// TwinCAT 3 PLC project _7000_Theresianum
// ProgramVersion: 3.1.4024.0
// libraries:
//   EfficientIO Communicator, * (EfficientIO)
//   EfficientIO ModbusTCP, * (EfficientIO)
//   Lynus Energy Basic, * (Lynus AG)
//   Lynus Persistent Data V1, * (Lynus AG)
//   Lynus Standards, * (Lynus AG)
//   Tc2_BABasic, * (Beckhoff Automation GmbH)
//   Tc2_Standard, * (Beckhoff Automation GmbH)
//   Tc2_System, * (Beckhoff Automation GmbH)
//   Tc2_Utilities, * (Beckhoff Automation GmbH)
//   Tc3_IotBase, * (Beckhoff Automation GmbH)
//   Tc3_JsonXml, * (Beckhoff Automation GmbH)
//   Tc3_Module, * (Beckhoff Automation GmbH)
// project tree:
//   / FastTask.TcTTO, MiddleTask.TcTTO, SlowTask.TcTTO
//   FBs/ FB_EM_Beckhoff_KL3403.TcPOU, FB_MqttCommunicator_V2_1.TcPOU, FB_Shelly_Pro.TcPOU (not stored), FB_Shelly_Pro1PM_Helper.TcPOU, FB_Shelly_Pro3EM.TcPOU, FB_Shelly_Pro3EM_Helper.TcPOU
//   POUs/ prgComEffIO.TcPOU, prgEM.TcPOU, prgPersistent.TcPOU, prgRWEffIO.TcPOU (not stored), prgShelly.TcPOU, prgVarEffIO.TcPOU (not stored), prg_SystemTime.TcPOU (not stored)
// real-time tasks:
//   TASK FastTask: cycle T#5ms, priority 6, ADS port 350
//   TASK MiddleTask: cycle T#10ms, priority 8, ADS port 351
//   TASK SlowTask: cycle T#20ms, priority 10, ADS port 352
// I/O:
//   DEVICE Gerät 1 (Beckhoff CCAT)
//   DEVICE Gerät 2 (CX-BK)
//     Box 1 (CX-BK)
// variable links:
//   (this object) <-> Device 2 (CX-BK)/Box 1 (CX-BK)
//     MiddleTask Inputs/prgEM.fbEM1.fbKL3403.byStateCH1 <-> Term 2 (KL3403)/Channel 1/Status
//     MiddleTask Inputs/prgEM.fbEM1.fbKL3403.byStateCH2 <-> Term 2 (KL3403)/Channel 2/Status
//     MiddleTask Inputs/prgEM.fbEM1.fbKL3403.byStateCH3 <-> Term 2 (KL3403)/Channel 3/Status
//     MiddleTask Inputs/prgEM.fbEM2.fbKL3403.byStateCH1 <-> Term 3 (KL3403)/Channel 1/Status
//     MiddleTask Inputs/prgEM.fbEM2.fbKL3403.byStateCH2 <-> Term 3 (KL3403)/Channel 2/Status
//     MiddleTask Inputs/prgEM.fbEM2.fbKL3403.byStateCH3 <-> Term 3 (KL3403)/Channel 3/Status
//     MiddleTask Inputs/prgEM.fbEM3.fbKL3403.byStateCH1 <-> Term 4 (KL3403)/Channel 1/Status
//     MiddleTask Inputs/prgEM.fbEM3.fbKL3403.byStateCH2 <-> Term 4 (KL3403)/Channel 2/Status
//     MiddleTask Inputs/prgEM.fbEM3.fbKL3403.byStateCH3 <-> Term 4 (KL3403)/Channel 3/Status
//     MiddleTask Inputs/prgEM.fbEM4.fbKL3403.byStateCH1 <-> Term 5 (KL3403)/Channel 1/Status
//     MiddleTask Inputs/prgEM.fbEM4.fbKL3403.byStateCH2 <-> Term 5 (KL3403)/Channel 2/Status
//     MiddleTask Inputs/prgEM.fbEM4.fbKL3403.byStateCH3 <-> Term 5 (KL3403)/Channel 3/Status
//     MiddleTask Inputs/prgEM.fbEM5.fbKL3403.byStateCH1 <-> Term 6 (KL3403)/Channel 1/Status
//     MiddleTask Inputs/prgEM.fbEM5.fbKL3403.byStateCH2 <-> Term 6 (KL3403)/Channel 2/Status
//     MiddleTask Inputs/prgEM.fbEM5.fbKL3403.byStateCH3 <-> Term 6 (KL3403)/Channel 3/Status
//     MiddleTask Inputs/prgEM.fbEM1.fbKL3403.iDataInCH1 <-> Term 2 (KL3403)/Channel 1/Daten Ein
//     MiddleTask Inputs/prgEM.fbEM1.fbKL3403.iDataInCH2 <-> Term 2 (KL3403)/Channel 2/Daten Ein
//     MiddleTask Inputs/prgEM.fbEM1.fbKL3403.iDataInCH3 <-> Term 2 (KL3403)/Channel 3/Daten Ein
//     MiddleTask Inputs/prgEM.fbEM2.fbKL3403.iDataInCH1 <-> Term 3 (KL3403)/Channel 1/Daten Ein
//     MiddleTask Inputs/prgEM.fbEM2.fbKL3403.iDataInCH2 <-> Term 3 (KL3403)/Channel 2/Daten Ein
//     MiddleTask Inputs/prgEM.fbEM2.fbKL3403.iDataInCH3 <-> Term 3 (KL3403)/Channel 3/Daten Ein
//     MiddleTask Inputs/prgEM.fbEM3.fbKL3403.iDataInCH1 <-> Term 4 (KL3403)/Channel 1/Daten Ein
//     MiddleTask Inputs/prgEM.fbEM3.fbKL3403.iDataInCH2 <-> Term 4 (KL3403)/Channel 2/Daten Ein
//     MiddleTask Inputs/prgEM.fbEM3.fbKL3403.iDataInCH3 <-> Term 4 (KL3403)/Channel 3/Daten Ein
//     MiddleTask Inputs/prgEM.fbEM4.fbKL3403.iDataInCH1 <-> Term 5 (KL3403)/Channel 1/Daten Ein
//     MiddleTask Inputs/prgEM.fbEM4.fbKL3403.iDataInCH2 <-> Term 5 (KL3403)/Channel 2/Daten Ein
//     MiddleTask Inputs/prgEM.fbEM4.fbKL3403.iDataInCH3 <-> Term 5 (KL3403)/Channel 3/Daten Ein
//     MiddleTask Inputs/prgEM.fbEM5.fbKL3403.iDataInCH1 <-> Term 6 (KL3403)/Channel 1/Daten Ein
//     MiddleTask Inputs/prgEM.fbEM5.fbKL3403.iDataInCH2 <-> Term 6 (KL3403)/Channel 2/Daten Ein
//     MiddleTask Inputs/prgEM.fbEM5.fbKL3403.iDataInCH3 <-> Term 6 (KL3403)/Channel 3/Daten Ein
//     MiddleTask Outputs/prgEM.fbEM1.fbKL3403.byCntrCH1 <-> Term 2 (KL3403)/Channel 1/Kontrolle
//     MiddleTask Outputs/prgEM.fbEM1.fbKL3403.byCntrCH2 <-> Term 2 (KL3403)/Channel 2/Kontrolle
//     MiddleTask Outputs/prgEM.fbEM1.fbKL3403.byCntrCH3 <-> Term 2 (KL3403)/Channel 3/Kontrolle
//     MiddleTask Outputs/prgEM.fbEM2.fbKL3403.byCntrCH1 <-> Term 3 (KL3403)/Channel 1/Kontrolle
//     MiddleTask Outputs/prgEM.fbEM2.fbKL3403.byCntrCH2 <-> Term 3 (KL3403)/Channel 2/Kontrolle
//     MiddleTask Outputs/prgEM.fbEM2.fbKL3403.byCntrCH3 <-> Term 3 (KL3403)/Channel 3/Kontrolle
//     MiddleTask Outputs/prgEM.fbEM3.fbKL3403.byCntrCH1 <-> Term 4 (KL3403)/Channel 1/Kontrolle
//     MiddleTask Outputs/prgEM.fbEM3.fbKL3403.byCntrCH2 <-> Term 4 (KL3403)/Channel 2/Kontrolle
//     MiddleTask Outputs/prgEM.fbEM3.fbKL3403.byCntrCH3 <-> Term 4 (KL3403)/Channel 3/Kontrolle
//     MiddleTask Outputs/prgEM.fbEM4.fbKL3403.byCntrCH1 <-> Term 5 (KL3403)/Channel 1/Kontrolle
//     MiddleTask Outputs/prgEM.fbEM4.fbKL3403.byCntrCH2 <-> Term 5 (KL3403)/Channel 2/Kontrolle
//     MiddleTask Outputs/prgEM.fbEM4.fbKL3403.byCntrCH3 <-> Term 5 (KL3403)/Channel 3/Kontrolle
//     MiddleTask Outputs/prgEM.fbEM5.fbKL3403.byCntrCH1 <-> Term 6 (KL3403)/Channel 1/Kontrolle
//     MiddleTask Outputs/prgEM.fbEM5.fbKL3403.byCntrCH2 <-> Term 6 (KL3403)/Channel 2/Kontrolle
//     MiddleTask Outputs/prgEM.fbEM5.fbKL3403.byCntrCH3 <-> Term 6 (KL3403)/Channel 3/Kontrolle

CONFIGURATION _7000_Theresianum
    RESOURCE PLC ON TwinCAT3
        TASK FastTask(INTERVAL := T#5ms, PRIORITY := 6);
        TASK MiddleTask(INTERVAL := T#10ms, PRIORITY := 8);
        TASK SlowTask(INTERVAL := T#20ms, PRIORITY := 10);
        PROGRAM prgVarEffIO WITH FastTask : prgVarEffIO;
        PROGRAM prgRWEffIO WITH FastTask : prgRWEffIO;
        PROGRAM prgPersistent WITH MiddleTask : prgPersistent;
        PROGRAM prgEM WITH MiddleTask : prgEM;
        PROGRAM prgShelly WITH MiddleTask : prgShelly;
        PROGRAM prgComEffIO WITH SlowTask : prgComEffIO;
    END_RESOURCE
END_CONFIGURATION

// ---- POUs/prgPersistent.TcPOU
PROGRAM prgPersistent
VAR
	fbUSV		: FB_WritePersistentData_CX81xx;
	fb_Reboot		: NT_reboot;
	m_Reboot		: BOOL:=FALSE;
END_VAR

fbUSV(
	eSaveModeData:= eUSVSaveMode.eSaveWhenPowerfail, 
	bLoadPersistentDataOk=> , 
	bPowerFailDetect=> , 
	bError=> , 
	bySaveProcess=> , 
	dwStorageLast24h=> , 
	udiErrorCode=> );
(*	
prg_SystemTime();

		
fb_Reboot(	netid := '',
			delay := 2,
			start := m_Reboot);
			
*)

END_PROGRAM

// ---- POUs/prgEM.TcPOU
PROGRAM prgEM
VAR
	fbKBusState					: FB_K_Bus_State;
	fbEM1						: FB_EM_Beckhoff_KL3403;			//Messung 1 Rest
	fbEM1Counter				: FB_EnergyCounter;
	fbEM2						: FB_EM_Beckhoff_KL3403;			//Messung 2 Schulküche
	fbEM2Counter				: FB_EnergyCounter;
	fbEM3						: FB_EM_Beckhoff_KL3403;			//Messung 3 Aufzüge
	fbEM3Counter				: FB_EnergyCounter;
	fbEM4						: FB_EM_Beckhoff_KL3403;			//Messung 4 Heizungsverteiler
	fbEM4Counter				: FB_EnergyCounter;
	fbEM5						: FB_EM_Beckhoff_KL3403;			//Messung 5 Verteiler 14 gesamt
	fbEM5Counter				: FB_EnergyCounter;
	
	lrPowerEM1_1				: LREAL;							//{#lynus.ag#()}
	lrPowerEM1_2				: LREAL;							//{#lynus.ag#()}
	lrPowerEM1_3				: LREAL;							//{#lynus.ag#()}
	lrPowerEM2_1				: LREAL;							//{#lynus.ag#()}
	lrPowerEM2_2				: LREAL;							//{#lynus.ag#()}
	lrPowerEM2_3				: LREAL;							//{#lynus.ag#()}
	lrPowerEM3_1				: LREAL;							//{#lynus.ag#()}
	lrPowerEM3_2				: LREAL;							//{#lynus.ag#()}
	lrPowerEM3_3				: LREAL;							//{#lynus.ag#()}
	lrPowerEM4_1				: LREAL;							//{#lynus.ag#()}
	lrPowerEM4_2				: LREAL;							//{#lynus.ag#()}
	lrPowerEM4_3				: LREAL;							//{#lynus.ag#()}
	lrPowerEM5_1				: LREAL;							//{#lynus.ag#()}
	lrPowerEM5_2				: LREAL;							//{#lynus.ag#()}
	lrPowerEM5_3				: LREAL;							//{#lynus.ag#()}
	
	lrPowerEM1_Total			: LREAL;							//{#lynus.ag#()}
	lrPowerEM2_Total			: LREAL;							//{#lynus.ag#()}
	lrPowerEM3_Total			: LREAL;							//{#lynus.ag#()}
	lrPowerEM4_Total			: LREAL;							//{#lynus.ag#()}
	lrPowerEM5_Total			: LREAL;							//{#lynus.ag#()}
	
	lrCounterGridCon			: LREAL;							
	//lrCounterGridProd			: LREAL;							
	
	lr_GridVoltage1_L1N_V		: LREAL;						
	lr_GridVoltage1_L2N_V		: LREAL;						
	lr_GridVoltage1_L3N_V		: LREAL;						
	lr_GridVoltage2_L1N_V		: LREAL;						
	lr_GridVoltage2_L2N_V		: LREAL;						
	lr_GridVoltage2_L3N_V		: LREAL;						
	lr_GridVoltage3_L1N_V		: LREAL;						
	lr_GridVoltage3_L2N_V		: LREAL;						
	lr_GridVoltage3_L3N_V		: LREAL;						
	lr_GridVoltage4_L1N_V		: LREAL;						
	lr_GridVoltage4_L2N_V		: LREAL;						
	lr_GridVoltage4_L3N_V		: LREAL;						
	lr_GridVoltage5_L1N_V		: LREAL;						
	lr_GridVoltage5_L2N_V		: LREAL;						
	lr_GridVoltage5_L3N_V		: LREAL;						

	lrReactivePowerGrid			: LREAL;							
	lrApparentPowerGrid			: LREAL;							
	
	lrPowerGrid					: LREAL;							//{#lynus.ag#()}

	lrPowerHouse				: LREAL;							//{#lynus.ag#()}
	tmp	: LREAL;
	tmp2	: LREAL;
END_VAR

VAR PERSISTENT
	
	lrCounterEM1					: LREAL;							//{#lynus.ag#()}
	lrCounterEM2					: LREAL;							//{#lynus.ag#()}
	lrCounterEM3					: LREAL;							//{#lynus.ag#()}
	lrCounterEM4					: LREAL;							//{#lynus.ag#()}
	lrCounterEM5					: LREAL;							//{#lynus.ag#()}

END_VAR

//The mapping of this function must be linked with the K-Bus State in the E/A Part
fbKBusState(	uiKBusState_OUT=> , 
				b_Kbus_notOk=> , 
				word_ErrorCount=> );
				
//The mapping of this function must be linked with the KL3403 in the E/A Part

fbEM1(										//Rest
	bEnable:= TRUE, 
	bChannel1Invers:= FALSE,				//Invert power data when transformer are mounted upside down
	bChannel2Invers:= FALSE,
	bChannel3Invers:= FALSE,
	uiCurrentTransformerRatioL1:= 400, 		//Transformer ratio on the secondary side
	uiCurrentTransformerRatioL2:= 400, 
	uiCurrentTransformerRatioL3:= 400, 
	uiKBusState_IN:= fbKBusState.uiKBusState_OUT, 
	stDataEMPower=> , 
	stDataEMCounter=> , 
	stDataEMPowerRealTime=> , 
	stDataEMCounterRealTime=> , 
	diNrOfEM_OUT=> );
	


fbEM2(										// Heizungsverteiler
	bEnable:= TRUE, 
	bChannel1Invers:= FALSE,				//Invert power data when transformer are mounted upside down
	bChannel2Invers:= FALSE,
	bChannel3Invers:= FALSE,	
	uiCurrentTransformerRatioL1:= 400, 		//Transformer ratio on the secondary side
	uiCurrentTransformerRatioL2:= 400, 
	uiCurrentTransformerRatioL3:= 400, 
	uiKBusState_IN:= fbKBusState.uiKBusState_OUT, 
	stDataEMPower=> , 
	stDataEMCounter=> , 
	stDataEMPowerRealTime=> , 
	stDataEMCounterRealTime=> , 
	diNrOfEM_OUT=> );
	
fbEM3(										// Aufzüge
	bEnable:= TRUE, 
	bChannel1Invers:= FALSE,				//Invert power data when transformer are mounted upside down
	bChannel2Invers:= FALSE,
	bChannel3Invers:= FALSE,
	uiCurrentTransformerRatioL1:= 300, 		//Transformer ratio on the secondary side
	uiCurrentTransformerRatioL2:= 300, 
	uiCurrentTransformerRatioL3:= 300, 
	uiKBusState_IN:= fbKBusState.uiKBusState_OUT, 
	stDataEMPower=> , 
	stDataEMCounter=> , 
	stDataEMPowerRealTime=> , 
	stDataEMCounterRealTime=> , 
	diNrOfEM_OUT=> );
	
fbEM4(										// Turnsaal
	bEnable:= TRUE, 
	bChannel1Invers:= FALSE,				//Invert power data when transformer are mounted upside down
	bChannel2Invers:= FALSE,
	bChannel3Invers:= FALSE,
	uiCurrentTransformerRatioL1:= 300, 		//Transformer ratio on the secondary side
	uiCurrentTransformerRatioL2:= 300, 
	uiCurrentTransformerRatioL3:= 300, 
	uiKBusState_IN:= fbKBusState.uiKBusState_OUT, 
	stDataEMPower=> , 
	stDataEMCounter=> , 
	stDataEMPowerRealTime=> , 
	stDataEMCounterRealTime=> , 
	diNrOfEM_OUT=> );
	
fbEM5(										// Verteiler Schulküchen (4x185mm2)
	bEnable:= TRUE, 
	bChannel1Invers:= FALSE,				//Invert power data when transformer are mounted upside down
	bChannel2Invers:= FALSE,
	bChannel3Invers:= FALSE,
	uiCurrentTransformerRatioL1:= 400, 		//Transformer ratio on the secondary side
	uiCurrentTransformerRatioL2:= 400, 
	uiCurrentTransformerRatioL3:= 400, 
	uiKBusState_IN:= fbKBusState.uiKBusState_OUT, 
	stDataEMPower=> , 
	stDataEMCounter=> , 
	stDataEMPowerRealTime=> , 
	stDataEMCounterRealTime=> , 
	diNrOfEM_OUT=> );

//lrCounterGridProd := fbEM1.stDataEMCounter.lrTotalCounterEnergy_Production;	

lrPowerEM1_1 := fbEM1.stDataEMPower.lrPowerL1;
lrPowerEM1_2 := fbEM1.stDataEMPower.lrPowerL2;
lrPowerEM1_3 := fbEM1.stDataEMPower.lrPowerL3;

lrPowerEM1_Total := fbEM1.stDataEMPower.lrPowerTotal;

lrReactivePowerGrid:=fbEM1.stDataEMPower.lrReactivePowerTotal;
lrApparentPowerGrid:=fbEM1.stDataEMPower.lrApparentPowerTotal;

lr_GridVoltage1_L1N_V:=fbEM1.stDataEMPower.lrVoltageL1N;
lr_GridVoltage1_L2N_V:=fbEM1.stDataEMPower.lrVoltageL2N;
lr_GridVoltage1_L3N_V:=fbEM1.stDataEMPower.lrVoltageL3N;

lrPowerEM2_1 := fbEM2.stDataEMPower.lrPowerL1;
lrPowerEM2_2 := fbEM2.stDataEMPower.lrPowerL2;
lrPowerEM2_3 := fbEM2.stDataEMPower.lrPowerL3;

lrPowerEM2_Total := fbEM2.stDataEMPower.lrPowerTotal;

lrReactivePowerGrid:=fbEM2.stDataEMPower.lrReactivePowerTotal;
lrApparentPowerGrid:=fbEM2.stDataEMPower.lrApparentPowerTotal;

lr_GridVoltage2_L1N_V:=fbEM2.stDataEMPower.lrVoltageL1N;
lr_GridVoltage2_L2N_V:=fbEM2.stDataEMPower.lrVoltageL2N;
lr_GridVoltage2_L3N_V:=fbEM2.stDataEMPower.lrVoltageL3N;

lrPowerEM3_1 := fbEM3.stDataEMPower.lrPowerL1;
lrPowerEM3_2 := fbEM3.stDataEMPower.lrPowerL2;
lrPowerEM3_3 := fbEM3.stDataEMPower.lrPowerL3;

lrPowerEM3_Total := fbEM3.stDataEMPower.lrPowerTotal;

lrReactivePowerGrid:=fbEM3.stDataEMPower.lrReactivePowerTotal;
lrApparentPowerGrid:=fbEM3.stDataEMPower.lrApparentPowerTotal;

lr_GridVoltage3_L1N_V:=fbEM3.stDataEMPower.lrVoltageL1N;
lr_GridVoltage3_L2N_V:=fbEM3.stDataEMPower.lrVoltageL2N;
lr_GridVoltage3_L3N_V:=fbEM3.stDataEMPower.lrVoltageL3N;

lrPowerEM4_1 := fbEM4.stDataEMPower.lrPowerL1;
lrPowerEM4_2 := fbEM4.stDataEMPower.lrPowerL2;
lrPowerEM4_3 := fbEM4.stDataEMPower.lrPowerL3;

lrPowerEM4_Total := fbEM4.stDataEMPower.lrPowerTotal;

lrReactivePowerGrid:=fbEM4.stDataEMPower.lrReactivePowerTotal;
lrApparentPowerGrid:=fbEM4.stDataEMPower.lrApparentPowerTotal;

lr_GridVoltage4_L1N_V:=fbEM4.stDataEMPower.lrVoltageL1N;
lr_GridVoltage4_L2N_V:=fbEM4.stDataEMPower.lrVoltageL2N;
lr_GridVoltage4_L3N_V:=fbEM4.stDataEMPower.lrVoltageL3N;

lrPowerEM5_1 := fbEM5.stDataEMPower.lrPowerL1;
lrPowerEM5_2 := fbEM5.stDataEMPower.lrPowerL2;
lrPowerEM5_3 := fbEM5.stDataEMPower.lrPowerL3;

lrPowerEM5_Total := fbEM5.stDataEMPower.lrPowerTotal;

lrReactivePowerGrid:=fbEM5.stDataEMPower.lrReactivePowerTotal;
lrApparentPowerGrid:=fbEM5.stDataEMPower.lrApparentPowerTotal;

lr_GridVoltage5_L1N_V:=fbEM5.stDataEMPower.lrVoltageL1N;
lr_GridVoltage5_L2N_V:=fbEM5.stDataEMPower.lrVoltageL2N;
lr_GridVoltage5_L3N_V:=fbEM5.stDataEMPower.lrVoltageL3N;

lrPowerGrid := LIMIT((fbEM1.stDataEMPower.lrPowerTotal + fbEM2.stDataEMPower.lrPowerTotal + fbEM3.stDataEMPower.lrPowerTotal + fbEM4.stDataEMPower.lrPowerTotal + fbEM5.stDataEMPower.lrPowerTotal),(fbEM1.stDataEMPower.lrPowerTotal + fbEM5.stDataEMPower.lrPowerTotal),999999);
tmp := fbEM1.stDataEMPower.lrPowerTotal + fbEM2.stDataEMPower.lrPowerTotal + fbEM3.stDataEMPower.lrPowerTotal + fbEM4.stDataEMPower.lrPowerTotal + fbEM5.stDataEMPower.lrPowerTotal;
tmp2 := fbEM1.stDataEMPower.lrPowerTotal + fbEM5.stDataEMPower.lrPowerTotal;

lrPowerHouse :=  lrPowerEM1_Total - (lrPowerEM2_Total + lrPowerEM3_Total + lrPowerEM4_Total);

lrCounterGridCon := fbEM1.stDataEMCounter.lrTotalCounterEnergy_Consumption + fbEM2.stDataEMCounter.lrTotalCounterEnergy_Consumption + fbEM3.stDataEMCounter.lrTotalCounterEnergy_Consumption + fbEM4.stDataEMCounter.lrTotalCounterEnergy_Consumption + fbEM5.stDataEMCounter.lrTotalCounterEnergy_Consumption;	
 
fbEM1Counter(
	byActiveTariff:= 1, 
	lrPowerInput:= lrPowerEM1_Total, 
	lrTotalCounterEnergy_Consumption=> , 
	lrTotalCounterEnergy_Production=> , 
	lrCounterEnergyT1_Consumption=> , 
	lrCounterEnergyT2_Consumption=> , 
	lrCounterEnergyT1_Production=> , 
	lrCounterEnergyT2_Production=> );
IF fbEM1Counter.lrTotalCounterEnergy_Consumption > lrCounterEM1 THEN  	
	lrCounterEM1 := fbEM1Counter.lrTotalCounterEnergy_Consumption;
END_IF

fbEM2Counter(
	byActiveTariff:= 1, 
	lrPowerInput:= lrPowerEM2_Total, 
	lrTotalCounterEnergy_Consumption=> , 
	lrTotalCounterEnergy_Production=> , 
	lrCounterEnergyT1_Consumption=> , 
	lrCounterEnergyT2_Consumption=> , 
	lrCounterEnergyT1_Production=> , 
	lrCounterEnergyT2_Production=> );
IF fbEM2Counter.lrTotalCounterEnergy_Consumption > lrCounterEM2 THEN  	
	lrCounterEM2 := fbEM2Counter.lrTotalCounterEnergy_Consumption;
END_IF

fbEM3Counter(
	byActiveTariff:= 1, 
	lrPowerInput:= lrPowerEM3_Total, 
	lrTotalCounterEnergy_Consumption=> , 
	lrTotalCounterEnergy_Production=> , 
	lrCounterEnergyT1_Consumption=> , 
	lrCounterEnergyT2_Consumption=> , 
	lrCounterEnergyT1_Production=> , 
	lrCounterEnergyT2_Production=> );
IF fbEM3Counter.lrTotalCounterEnergy_Consumption > lrCounterEM3 THEN  	
	lrCounterEM3 := fbEM3Counter.lrTotalCounterEnergy_Consumption;
END_IF

fbEM4Counter(
	byActiveTariff:= 1, 
	lrPowerInput:= lrPowerEM4_Total, 
	lrTotalCounterEnergy_Consumption=> , 
	lrTotalCounterEnergy_Production=> , 
	lrCounterEnergyT1_Consumption=> , 
	lrCounterEnergyT2_Consumption=> , 
	lrCounterEnergyT1_Production=> , 
	lrCounterEnergyT2_Production=> );
IF fbEM4Counter.lrTotalCounterEnergy_Consumption > lrCounterEM4 THEN  	
	lrCounterEM4 := fbEM4Counter.lrTotalCounterEnergy_Consumption;
END_IF
 
 fbEM5Counter(
	byActiveTariff:= 1, 
	lrPowerInput:= lrPowerEM5_Total, 
	lrTotalCounterEnergy_Consumption=> , 
	lrTotalCounterEnergy_Production=> , 
	lrCounterEnergyT1_Consumption=> , 
	lrCounterEnergyT2_Consumption=> , 
	lrCounterEnergyT1_Production=> , 
	lrCounterEnergyT2_Production=> );
IF fbEM5Counter.lrTotalCounterEnergy_Consumption > lrCounterEM5 THEN  	
	lrCounterEM5 := fbEM5Counter.lrTotalCounterEnergy_Consumption;
END_IF

END_PROGRAM

// ---- FBs/FB_EM_Beckhoff_KL3403.TcPOU
FUNCTION_BLOCK FB_EM_Beckhoff_KL3403
VAR_INPUT PERSISTENT
	bEnable							: BOOL;											//Enable the function
	bChannel1Invers					: BOOL;											//Invert the Output data from Channel 1. = L1
	bChannel2Invers					: BOOL;											//Invert the Output data from Channel 2. = L2
	bChannel3Invers					: BOOL;											//Invert the Output data from Channel 3. = L3
	uiCurrentTransformerRatioL1		: UINT;											//Current Transformer Ratio for Channel 1 (L1)
	uiCurrentTransformerRatioL2		: UINT;											//Current Transformer Ratio for Channel 2 (L2)
	uiCurrentTransformerRatioL3		: UINT;											//Current Transformer Ratio for Channel 3 (L3)
END_VAR
VAR_INPUT
	uiKBusState_IN					: UINT;											//K-Bus State from the K-Bus Box on wich the Terminal is connected. (Connect with FB_K_Bus_state)
END_VAR
VAR_OUTPUT
	stDataEMPower					: ST_ElectricMeter_Output_Power;				//Output structure with Data from Electric Meter (Power Data)
	stDataEMCounter					: ST_ElectricMeter_Output_Counter;				//Output structure with Data from Electric Meter (Counter Data)
	stDataEMPowerRealTime			: ST_ElectricMeter_Output_Power;				//Output structure with Data from Electric Meter (Power Data RealTime)
	stDataEMCounterRealTime			: ST_ElectricMeter_Output_Counter;				//Output structure with Data from Electric Meter (Counter Data RealTime)
	diNrOfEM_OUT					: DINT;											//Active Number from the Electric Meter for using on other functions
END_VAR
VAR
	{attribute 'conditionalshow'}
	fbEM							: FB_ElectricMeter;								//Electric Meter Function
	{attribute 'conditionalshow'}
	fbEnergyCounter					: FB_EnergyCounter;								//FB energy Counter, because the KL3403 has no nice logic for the Energy value
	{attribute 'hide'}
	fbNumberDevice					: FB_NumberOfDevice;							//Function block to calcualte the number of the Device
	fbKL3403						: FB_KL3403_SimpleProcessImage;					//Function KL3403
	{attribute 'hide'}
	stDataL1						: ST_KL3403;									//Data from Channel 1 (L1)
	{attribute 'hide'}
	stDataL2						: ST_KL3403;									//Data from Channel 2 (L2)
	{attribute 'hide'}
	stDataL3						: ST_KL3403;									//Data from Channel 3 (L3)
	{attribute 'hide'}
	timDissableFunctions			: TON;											//Timer to dissable the Function after Lynus_Standards.Constants_General.tTimeDissableLynusFunctions Days without connection to the Lynus Cloud
	{attribute 'hide'}
	timResetConnectionOnGVL			: TON;											//Timer to try reset the connection Flag on the GVL. (When somebody delete the Connection Function and make only a onlinechange)
	{attribute 'hide'}
	timSetCounterValues				: TON;											//Timer to set the counter values from the KL3403 Function to the EM Function
	{attribute 'hide'}
	arrPD							: ARRAY[1..7] OF FB_PersistentData_Number;		//Function to save persistent data
	{attribute 'hide'}
	byWaitInStep					: BYTE;											//Wait in Step before start to clean data on PLC
	{attribute 'hide'}
	iStateGVLData					: INT;											//State machine to handle the data on the GVL
	{attribute 'hide'}
	diCounterForGVL					: DINT;											//Counter to clean old data on GVL
END_VAR

//Creator : Kai Ebensperger
//Company : Lynus AG
//Date : 04.10.2021
//Version : 1.0.0.0

//Stefan: Addes S and Q calculation

//With this function is possible to read out all Information from a KL3403
//This Function support only the Simple Process Image and the Ratio in the Terminal register must be Set allways to 1.

//NOTE for diNr.....Designation => 
//_IN = Here Data come in from other Functions or go out to other functions about the GVL
//_OUT = Here Data go out to other functions about the GVL

(*-------------------------------------------------------------Calcualte the number of EM---------------------------------------------------------------*)

fbNumberDevice(
	diActualNumberOfDevices:= Lynus_Standards.GVL_Energy.stNumberOfDevices.diNumberOfElectricMeters, 
	diMaxNumberOfDevices:= Constants_Energy.diMaxNumberOfElectricMeters, 
	udiCounterOnlineChange:= TwinCAT_SystemInfoVarList._AppInfo.OnlineChangeCnt, 
	bNumberIsCalculatet=> , 
	bFPNumberIsCalculatet=> , 
	bOnlineChange=> , 
	diNumberForThisDevice=> diNrOfEM_OUT, 
	diNumberOfTotalDevices=> );

//Write new Numer on GVL
IF fbNumberDevice.bFPNumberIsCalculatet THEN
	Lynus_Standards.GVL_Energy.stNumberOfDevices.diNumberOfElectricMeters := fbNumberDevice.diNumberOfTotalDevices;	
END_IF

//Delete old Number on GVL
IF fbNumberDevice.bOnlineChange THEN 
	Lynus_Standards.GVL_Energy.stNumberOfDevices.diNumberOfElectricMeters := diNrOfEM_OUT;	
		iStateGVLData := 1; 
END_IF

(*-------------------------------------------------------------Service from Backend is ready and check the connection to backen for dissabel/enable Function---------------------------------------------------------------*)

//Try to reset the variable for connection on the GVL. When all is normal then the Lynus Mqtt connection function set this variable to true in the next cycle
//When we have no connection to the backend then after Lynus_Standards.Constants_General.tTimeDissableLynusFunctions days the Function is dissabled with all of his functionalities
timResetConnectionOnGVL(IN:= NOT timResetConnectionOnGVL.Q, PT:= T#1H, Q=> , ET=> );
	IF timResetConnectionOnGVL.Q THEN Lynus_Standards.GVL_Communicator.bStateConnectionToEnableFunctions := FALSE; END_IF
		IF NOT Lynus_Standards.GVL_Communicator.bStateConnectionToEnableFunctions THEN timDissableFunctions.IN := TRUE; ELSE timDissableFunctions.IN := FALSE; END_IF  
			timDissableFunctions(IN:= , PT:= Lynus_Standards.Constants_General.tTimeDissableLynusFunctions, Q=> , ET=> );

(*----------------------------------------------------------------------------------------KL3403 Communication----------------------------------------------------------------------------------------------*)

fbKL3403(
	uiKBusState_IN:= uiKBusState_IN, 
	uiCurrentTransformerRatioL1:= uiCurrentTransformerRatioL1,
	uiCurrentTransformerRatioL2:= uiCurrentTransformerRatioL2,
	uiCurrentTransformerRatioL3:= uiCurrentTransformerRatioL3,
	rResolutionCurrent:= 0.001,
	rResolutionPower:= 0.1,
	rResolutionEnergy:= 0.01,
	stDataL1=> , 
	stDataL2=> ,
	stDataL3=> );

//Invert the Output data, because it is possible that the current transformers have been mounted in different mounting positions.
IF NOT bChannel1Invers THEN
	stDataL1 := fbKL3403.stDataL1;
ELSE
	stDataL1.byErrorWarning := fbKL3403.stDataL1.byErrorWarning;
	stDataL1.rCurrent := fbKL3403.stDataL1.rCurrent;
	stDataL1.rVoltage := fbKL3403.stDataL1.rVoltage;
	stDataL1.rPower := fbKL3403.stDataL1.rPower * - 1;
	stDataL1.rPowerfactor := fbKL3403.stDataL1.rPowerfactor;
	stDataL1.rEnergy := fbKL3403.stDataL1.rEnergy;
	stDataL1.rFrequency := fbKL3403.stDataL1.rFrequency;
	stDataL1.rPeakValueCurrent := fbKL3403.stDataL1.rPeakValueCurrent;
	stDataL1.rPeakValueVoltage := fbKL3403.stDataL1.rPeakValueVoltage;
	stDataL1.rPeakValuePower := fbKL3403.stDataL1.rPeakValuePower * - 1;
	stDataL1.rMinValueCurrent := fbKL3403.stDataL1.rMinValueCurrent;
	stDataL1.rMinValueVoltage := fbKL3403.stDataL1.rMinValueVoltage;
	stDataL1.rMinValuePower := fbKL3403.stDataL1.rMinValuePower * - 1;
END_IF

IF NOT bChannel2Invers THEN
	stDataL2 := fbKL3403.stDataL2;
ELSE
	stDataL2.byErrorWarning := fbKL3403.stDataL2.byErrorWarning;
	stDataL2.rCurrent := fbKL3403.stDataL2.rCurrent;
	stDataL2.rVoltage := fbKL3403.stDataL2.rVoltage;
	stDataL2.rPower := fbKL3403.stDataL2.rPower * - 1;
	stDataL2.rPowerfactor := fbKL3403.stDataL2.rPowerfactor;
	stDataL2.rEnergy := fbKL3403.stDataL2.rEnergy;
	stDataL2.rFrequency := fbKL3403.stDataL2.rFrequency;
	stDataL2.rPeakValueCurrent := fbKL3403.stDataL2.rPeakValueCurrent;
	stDataL2.rPeakValueVoltage := fbKL3403.stDataL2.rPeakValueVoltage;
	stDataL2.rPeakValuePower := fbKL3403.stDataL2.rPeakValuePower * - 1;
	stDataL2.rMinValueCurrent := fbKL3403.stDataL2.rMinValueCurrent;
	stDataL2.rMinValueVoltage := fbKL3403.stDataL2.rMinValueVoltage;
	stDataL2.rMinValuePower := fbKL3403.stDataL2.rMinValuePower * - 1;
END_IF

IF NOT bChannel3Invers THEN
	stDataL3 := fbKL3403.stDataL3;
ELSE
	stDataL3.byErrorWarning := fbKL3403.stDataL3.byErrorWarning;
	stDataL3.rCurrent := fbKL3403.stDataL3.rCurrent;
	stDataL3.rVoltage := fbKL3403.stDataL3.rVoltage;
	stDataL3.rPower := fbKL3403.stDataL3.rPower * - 1;
	stDataL3.rPowerfactor := fbKL3403.stDataL3.rPowerfactor;
	stDataL3.rEnergy := fbKL3403.stDataL3.rEnergy;
	stDataL3.rFrequency := fbKL3403.stDataL3.rFrequency;
	stDataL3.rPeakValueCurrent := fbKL3403.stDataL3.rPeakValueCurrent;
	stDataL3.rPeakValueVoltage := fbKL3403.stDataL3.rPeakValueVoltage;
	stDataL3.rPeakValuePower := fbKL3403.stDataL3.rPeakValuePower * - 1;
	stDataL3.rMinValueCurrent := fbKL3403.stDataL3.rMinValueCurrent;
	stDataL3.rMinValueVoltage := fbKL3403.stDataL3.rMinValueVoltage;
	stDataL3.rMinValuePower := fbKL3403.stDataL3.rMinValuePower * - 1;
END_IF
	
(*----------------------------------------------------------------------------------------Energy Counter Function----------------------------------------------------------------------------------------------*)

//For the KL3403 we use a external Energy Counter Function. So we can count Import and Export Energy with the KL3403.
//Attetntion, the KL3403 is not MID Conform. Thus, these values must not be used for billing.
fbEnergyCounter(
	byActiveTariff:= 1, 
	lrPowerInput:= (stDataL1.rPower + stDataL2.rPower + stDataL3.rPower) / 1000, 
	lrTotalCounterEnergy_Consumption=> , 
	lrTotalCounterEnergy_Production=> , 
	lrCounterEnergyT1_Consumption=> , 
	lrCounterEnergyT2_Consumption=> , 
	lrCounterEnergyT1_Production=> , 
	lrCounterEnergyT2_Production=> );

(*----------------------------------------------------------------------------------------Electric Meter Function----------------------------------------------------------------------------------------------*)

//Error
IF timDissableFunctions.Q THEN fbEM.bWarning := TRUE; fbEM.iWarningCode := 0; ELSE fbEM.bWarning := FALSE; END_IF 
	IF Lynus_Standards.GVL_Energy.stNumberOfDevices.diNumberOfElectricMeters > Constants_Energy.diMaxNumberOfElectricMeters OR 
		stDataL1.byErrorWarning = 2 OR stDataL2.byErrorWarning = 2 OR stDataL3.byErrorWarning = 2 THEN 
			fbEM.bError := TRUE; 
	ELSE 
			fbEM.bError := FALSE; 
	END_IF
		IF Lynus_Standards.GVL_Energy.stNumberOfDevices.diNumberOfElectricMeters > Constants_Energy.diMaxNumberOfElectricMeters THEN fbEM.iErrorCode := 1;
		ELSIF stDataL1.byErrorWarning = 2 OR stDataL2.byErrorWarning = 2 OR stDataL3.byErrorWarning = 2 THEN fbEM.iErrorCode := 0;
		END_IF

timSetCounterValues(IN:= bEnable AND NOT timSetCounterValues.Q, PT:= T#2S, Q=> , ET=> );		

//Function
fbEM(
	bEnable:= bEnable AND NOT timDissableFunctions.Q, 
	bError:= , 
	bEnableReadOutFunction:= FALSE, 
	bWriteWithDelay:= TRUE, 
	bPowerDataInvers:= FALSE,
	bReadOutDataDone:= timSetCounterValues.Q,
	iTimeReadOutInterval:= 0, 
	iErrorCode:= , 
	iWarningCode:= , 
	lrTotalCounterEnergy_Consumption:= fbEnergyCounter.lrTotalCounterEnergy_Consumption,
	lrTotalCounterEnergy_Production:= fbEnergyCounter.lrTotalCounterEnergy_Production, 
	lrCounterEnergyT1_Consumption:= fbEnergyCounter.lrCounterEnergyT1_Consumption,
	lrCounterEnergyT2_Consumption:= fbEnergyCounter.lrCounterEnergyT2_Consumption,
	lrCounterEnergyT1_Production:= fbEnergyCounter.lrCounterEnergyT1_Production, 
	lrCounterEnergyT2_Production:= fbEnergyCounter.lrCounterEnergyT2_Production, 
	lrCurrentL1:= stDataL1.rCurrent, 
	lrVoltageL1N:= stDataL1.rVoltage, 
	lrVoltageL1L2:= stDataL1.rVoltage*SQRT(3), 
	lrPowerL1:= stDataL1.rPower, 
	lrCurrentL2:= stDataL2.rCurrent, 
	lrVoltageL2N:= stDataL2.rVoltage, 
	lrVoltageL2L3:= stDataL2.rVoltage*SQRT(3), 
	lrPowerL2:= stDataL2.rPower, 
	lrCurrentL3:= stDataL3.rCurrent, 
	lrVoltageL3N:= stDataL3.rVoltage, 
	lrVoltageL3L1:= stDataL3.rVoltage*SQRT(3), 
	lrPowerL3:= stDataL3.rPower, 
	lrPowerTotal:= stDataL1.rPower + stDataL2.rPower + stDataL3.rPower, 
	lrFrequency:= (stDataL1.rFrequency + stDataL2.rFrequency + stDataL3.rFrequency) / 3, 
 	lrApparentPowerTotal:=,
	lrReactivePowerTotal:=, 
	tTimDelayOutput:= T#5S, 
	stDataEMOutPower=> stDataEMPowerRealTime, 
	stDataEMOutPowerDelay=> stDataEMPower, 
	stDataEMOutCounter=> stDataEMCounterRealTime,
	stDataEMOutCounterDelay=> stDataEMCounter,
	bReadOutMeter=> );
(*
	IF  stDataL1.rPowerfactor <>0 AND stDataL2.rPowerfactor <>0 AND stDataL3.rPowerfactor <>0 THEN
		fbEM.lrApparentPowerTotal:= ABS(stDataL1.rPower)/ABS(stDataL1.rPowerfactor) + ABS(stDataL2.rPower)/ABS(stDataL2.rPowerfactor) + ABS(stDataL3.rPower)/ABS(stDataL3.rPowerfactor); 
	END_IF	
*)


	//calculate total apparant power in VA
	fbEM.lrApparentPowerTotal := fbEM.lrVoltageL1N * fbEM.lrCurrentL1 + fbEM.lrVoltageL2N * fbEM.lrCurrentL2 +  fbEM.lrVoltageL3N * fbEM.lrCurrentL3;
	
	IF fbEM.lrApparentPowerTotal<>0 AND fbEM.lrPowerTotal<>0 AND fbEM.lrApparentPowerTotal> fbEM.lrPowerTotal THEN
		fbEM.lrReactivePowerTotal:= SQRT(ABS(fbEM.lrApparentPowerTotal*fbEM.lrApparentPowerTotal - ABS(fbEM.lrPowerTotal*fbEM.lrPowerTotal)));	
	END_IF
	IF stDataL1.rPowerfactor<>0 AND stDataL2.rPowerfactor <>0 AND stDataL3.rPowerfactor<>0 THEN 	// check that not all cos phi are not 0
		IF (stDataL1.rPowerfactor+stDataL2.rPowerfactor+stDataL3.rPowerfactor)<>0 THEN				// check that the sum is not 0	
			IF 	(stDataL1.rPowerfactor+stDataL2.rPowerfactor+stDataL3.rPowerfactor)/3<0 THEN		// check is the average is below 0 / capacitive
				fbEM.lrReactivePowerTotal:=fbEM.lrReactivePowerTotal*(-1);
			END_IF
		END_IF	
	END_IF
(*-----------------------------------------------------------Handle data to Global structure for Electric Meter-----------------------------------------------------------------*)

CASE iStateGVLData OF
	
	0://Init Step
		byWaitInStep := 0;
			diCounterForGVL := 1;
	
	1://Wait for 4 Steps before clean al Data on GVL
		byWaitInStep := byWaitInStep + 1;
			IF byWaitInStep >= 4 AND fbNumberDevice.bNumberIsCalculatet THEN iStateGVLData := 2; END_IF
				//To much Devices, back to the Init step
				IF byWaitInStep >= 4 AND NOT fbNumberDevice.bNumberIsCalculatet THEN iStateGVLData := 0; END_IF	
			
	2://Clear all Data in GVL
		Lynus_Standards.GVL_Energy.stDataElectricMeters[diCounterForGVL].bEnabled := FALSE;	
			Lynus_Standards.GVL_Energy.stDataElectricMeters[diCounterForGVL].byErrorWarning := 0;
				Lynus_Standards.GVL_Energy.stDataElectricMeters[diCounterForGVL].lrCounterEnergyT1_Consumption := 0;
					Lynus_Standards.GVL_Energy.stDataElectricMeters[diCounterForGVL].lrCounterEnergyT1_Production := 0;
						Lynus_Standards.GVL_Energy.stDataElectricMeters[diCounterForGVL].lrCounterEnergyT2_Consumption := 0;
							Lynus_Standards.GVL_Energy.stDataElectricMeters[diCounterForGVL].lrCounterEnergyT2_Production := 0;
								Lynus_Standards.GVL_Energy.stDataElectricMeters[diCounterForGVL].lrPower := 0;
									Lynus_Standards.GVL_Energy.stDataElectricMeters[diCounterForGVL].lrPowerConsumption := 0;
										Lynus_Standards.GVL_Energy.stDataElectricMeters[diCounterForGVL].lrPowerProduction := 0;
											Lynus_Standards.GVL_Energy.stDataElectricMeters[diCounterForGVL].lrTotalCounterEnergy_Consumption := 0;
												Lynus_Standards.GVL_Energy.stDataElectricMeters[diCounterForGVL].lrTotalCounterEnergy_Production := 0;
		
		//Electric Meters
		diCounterForGVL := diCounterForGVL + 1;
			diCounterForGVL := LIMIT(0,diCounterForGVL,Constants_Energy.diMaxNumberOfElectricMeters);
				//Back to the init step
				IF diCounterForGVL >= Constants_Energy.diMaxNumberOfElectricMeters THEN iStateGVLData := 0; END_IF

END_CASE 	 

//Write Data on GVL for Electric Meter
IF diNrOfEM_OUT > 0 AND fbNumberDevice.bNumberIsCalculatet THEN
	Lynus_Standards.GVL_Energy.stDataElectricMeters[diNrOfEM_OUT].bEnabled := fbEM.stDataEMOutPower.bEnabled;
		Lynus_Standards.GVL_Energy.stDataElectricMeters[diNrOfEM_OUT].byErrorWarning := fbEM.stDataEMOutPower.byErrorWarning;
			Lynus_Standards.GVL_Energy.stDataElectricMeters[diNrOfEM_OUT].lrCounterEnergyT1_Consumption := fbEM.stDataEMOutCounter.lrCounterEnergyT1_Consumption;
				Lynus_Standards.GVL_Energy.stDataElectricMeters[diNrOfEM_OUT].lrCounterEnergyT1_Production := fbEM.stDataEMOutCounter.lrCounterEnergyT1_Production;
					Lynus_Standards.GVL_Energy.stDataElectricMeters[diNrOfEM_OUT].lrCounterEnergyT2_Consumption := fbEM.stDataEMOutCounter.lrCounterEnergyT2_Consumption;
						Lynus_Standards.GVL_Energy.stDataElectricMeters[diNrOfEM_OUT].lrCounterEnergyT2_Production := fbEM.stDataEMOutCounter.lrCounterEnergyT2_Production;		
							Lynus_Standards.GVL_Energy.stDataElectricMeters[diNrOfEM_OUT].lrPower := fbEM.stDataEMOutPower.lrPowerTotal;
								Lynus_Standards.GVL_Energy.stDataElectricMeters[diNrOfEM_OUT].lrPowerConsumption := fbEM.stDataEMOutPower.lrPowerConsumption;
									Lynus_Standards.GVL_Energy.stDataElectricMeters[diNrOfEM_OUT].lrPowerProduction := fbEM.stDataEMOutPower.lrPowerProduction;
										Lynus_Standards.GVL_Energy.stDataElectricMeters[diNrOfEM_OUT].lrTotalCounterEnergy_Consumption := fbEM.stDataEMOutCounter.lrTotalCounterEnergy_Consumption;
											Lynus_Standards.GVL_Energy.stDataElectricMeters[diNrOfEM_OUT].lrTotalCounterEnergy_Production := fbEM.stDataEMOutCounter.lrTotalCounterEnergy_Production;
END_IF

(*----------------------------------------------------------Save persistent data----------------------------------------------------------------*)

arrPD[1](lrValue:= BOOL_TO_LREAL(bEnable), bEventBasedActive=> );
arrPD[2](lrValue:= UINT_TO_LREAL(uiCurrentTransformerRatioL1), bEventBasedActive=> );
arrPD[3](lrValue:= UINT_TO_LREAL(uiCurrentTransformerRatioL2), bEventBasedActive=> );
arrPD[4](lrValue:= UINT_TO_LREAL(uiCurrentTransformerRatioL3), bEventBasedActive=> );
arrPD[5](lrValue:= BOOL_TO_LREAL(bChannel1Invers), bEventBasedActive=> );
arrPD[6](lrValue:= BOOL_TO_LREAL(bChannel2Invers), bEventBasedActive=> );
arrPD[7](lrValue:= BOOL_TO_LREAL(bChannel3Invers), bEventBasedActive=> );

END_FUNCTION_BLOCK

// ---- POUs/prgShelly.TcPOU
PROGRAM prgShelly
VAR
// Theresianum, Diverse Steckdosen
	fbShelly1					: FB_Shelly_Pro3EM;	
	lrPowerTotal_Shelly1		: LREAL;
	lrPowerTotal_Shelly1_kW		: LREAL;			//{#lynus.ag#()}
	
	//Messung 2, Patchkasten, EDV-Steckdosen
	
	fbShelly2					: FB_Shelly_Pro3EM;	
	lrPowerTotal_Shelly2		: LREAL;
	lrPowerTotal_Shelly2_kW		: LREAL;			//{#lynus.ag#()}
	
	//Messung 3, Klausur KG
	
	fbShelly3					: FB_Shelly_Pro3EM;	
	lrPowerTotal_Shelly3		: LREAL;
	lrPowerTotal_Shelly3_kW		: LREAL;			//{#lynus.ag#()}
	
	//Messung 4, Klausur EG
	
	fbShelly4					: FB_Shelly_Pro3EM;	
	lrPowerTotal_Shelly4		: LREAL;
	lrPowerTotal_Shelly4_kW		: LREAL;			//{#lynus.ag#()}

	//Messung 5, Klausur ZWG
	
	fbShelly5					: FB_Shelly_Pro3EM;	
	lrPowerTotal_Shelly5		: LREAL;
	lrPowerTotal_Shelly5_kW		: LREAL;			//{#lynus.ag#()}
	
	//Messung 6, Klausur OG
	
	fbShelly6					: FB_Shelly_Pro3EM;	
	lrPowerTotal_Shelly6		: LREAL;
	lrPowerTotal_Shelly6_kW		: LREAL;			//{#lynus.ag#()}
	
	//Messung 7, Klausur F27
	
	fbShelly7					: FB_Shelly_Pro3EM;	
	lrPowerTotal_Shelly7		: LREAL;
	lrPowerTotal_Shelly7_kW		: LREAL;			//{#lynus.ag#()}
	
	//Messung 8, Klausur F28
	
	fbShelly8					: FB_Shelly_Pro3EM;	
	lrPowerTotal_Shelly8		: LREAL;
	lrPowerTotal_Shelly8_kW		: LREAL;			//{#lynus.ag#()}

	//Messung 9
	
	fbShelly9					: FB_Shelly_Pro3EM;	
	lrPowerTotal_Shelly9		: LREAL;
	lrPowerTotal_Shelly9_kW		: LREAL;			//{#lynus.ag#()}
	
	//Messung 10
	
	fbShelly10					: FB_Shelly_Pro3EM;	
	lrPowerTotal_Shelly10		: LREAL;
	lrPowerTotal_Shelly10_kW	: LREAL;			//{#lynus.ag#()}
	
	//Messung 11
	
	fbShelly11					: FB_Shelly_Pro3EM;
	lrPowerTotal_Shelly11		: LREAL;
	lrPowerTotal_Shelly11_kW	: LREAL;			//{#lynus.ag#()}
	
	//Messung 12
	
	fbShelly12					: FB_Shelly_Pro3EM;	
	lrPowerTotal_Shelly12		: LREAL;
	lrPowerTotal_Shelly12_kW	: LREAL;			//{#lynus.ag#()}
	
	// other
	
	lrPowerV16_Kitchen_kW		: LREAL;			//{#lynus.ag#()}
	fbKitchenCounter			: FB_EnergyCounter;
	

END_VAR

VAR PERSISTENT
	
// trigger command execution
	bEnable_Shelly1				: BOOL:=TRUE;				//{#lynus.ag#()}
	bEnable_Shelly2				: BOOL:=TRUE;				//{#lynus.ag#()}
	bEnable_Shelly3				: BOOL:=TRUE;				//{#lynus.ag#()}
	bEnable_Shelly4				: BOOL:=TRUE;				//{#lynus.ag#()}
	bEnable_Shelly5				: BOOL:=TRUE;				//{#lynus.ag#()}
	bEnable_Shelly6				: BOOL:=TRUE;				//{#lynus.ag#()}
	bEnable_Shelly7				: BOOL:=TRUE;				//{#lynus.ag#()}
	bEnable_Shelly8				: BOOL:=TRUE;				//{#lynus.ag#()}
	bEnable_Shelly9				: BOOL:=TRUE;				//{#lynus.ag#()}
	bEnable_Shelly10			: BOOL:=FALSE;				//{#lynus.ag#()}
	bEnable_Shelly11			: BOOL:=FALSE;				//{#lynus.ag#()}
	bEnable_Shelly12			: BOOL:=FALSE;				//{#lynus.ag#()}
	
	lrCounterKitchen			: LREAL;					//{#lynus.ag#()}
	
END_VAR

// Grid Div 3-phase, 400V
fbShelly1(
	bStart:= bEnable_Shelly1, 
	tDelayRequest:= T#20S, 
	sHostname:= '192.168.178.210', 
	bValidResult=> , 
	bBusy=> , 
	bError=> , 
	bDone=> , 
	hrErrorCode=> ,
	lrpowertotal=> lrPowerTotal_Shelly1);

// re-calc to kW
lrPowerTotal_Shelly1_kW := lrPowerTotal_Shelly1 / 1000;

fbShelly2(
	bStart:= bEnable_Shelly2, 
	tDelayRequest:= T#20S, 
	sHostname:= '192.168.178.211', 
	bValidResult=> , 
	bBusy=> , 
	bError=> , 
	bDone=> , 
	hrErrorCode=> ,
	lrPowerTotal=> lrPowerTotal_Shelly2);

// re-calc to kW
lrPowerTotal_Shelly2_kW := lrPowerTotal_Shelly2 / 1000;

fbShelly3(							//UV9 F11
	bStart:= bEnable_Shelly3, 
	tDelayRequest:= T#20S, 
	sHostname:= '192.168.178.212', 
	bValidResult=> , 
	bBusy=> , 
	bError=> , 
	bDone=> , 
	hrErrorCode=> ,
	lrPowerTotal=> lrPowerTotal_Shelly3);
// re-calc to kW
lrPowerTotal_Shelly3_kW := lrPowerTotal_Shelly3 / 1000;

fbShelly4(							//UV9 F21
	bStart:= bEnable_Shelly4, 
	tDelayRequest:= T#20S, 
	sHostname:= '192.168.178.213', 
	bValidResult=> , 
	bBusy=> , 
	bError=> , 
	bDone=> , 
	hrErrorCode=> ,
	lrPowerTotal=> lrPowerTotal_Shelly4);

// re-calc to kW
lrPowerTotal_Shelly4_kW := lrPowerTotal_Shelly4 / 1000;

fbShelly5(							//UV9 F31
	bStart:= bEnable_Shelly5, 
	tDelayRequest:= T#20S, 
	sHostname:= '192.168.178.214', 
	bValidResult=> , 
	bBusy=> , 
	bError=> , 
	bDone=> , 
	hrErrorCode=> ,
	lrPowerTotal=> lrPowerTotal_Shelly5);

// re-calc to kW
lrPowerTotal_Shelly5_kW := lrPowerTotal_Shelly5 / 1000;

fbShelly6(						//UV9 F41 
	bStart:= bEnable_Shelly6, 
	tDelayRequest:= T#20S, 
	sHostname:= '192.168.178.215', 
	bValidResult=> , 
	bBusy=> , 
	bError=> , 
	bDone=> , 
	hrErrorCode=> ,
	lrPowerTotal=> lrPowerTotal_Shelly6);

// re-calc to kW
lrPowerTotal_Shelly6_kW := lrPowerTotal_Shelly6 / 1000;

fbShelly7(						//UV16 F28
	bStart:= bEnable_Shelly7, 
	tDelayRequest:= T#20S, 
	sHostname:= '192.168.178.216', 
	bValidResult=> , 
	bBusy=> , 
	bError=> , 
	bDone=> , 
	hrErrorCode=> ,
	lrPowerTotal=> lrPowerTotal_Shelly7);

// re-calc to kW
lrPowerTotal_Shelly7_kW := lrPowerTotal_Shelly7 / -1000; //Invertiert

fbShelly8(						//UV16 F29
	bStart:= bEnable_Shelly8, 
	tDelayRequest:= T#20S, 
	sHostname:= '192.168.178.217', 
	bValidResult=> , 
	bBusy=> , 
	bError=> , 
	bDone=> , 
	hrErrorCode=> ,
	lrPowerTotal=> lrPowerTotal_Shelly8);

// re-calc to kW
lrPowerTotal_Shelly8_kW := lrPowerTotal_Shelly8 / 1000;

fbShelly9(						//UV16 F30
	bStart:= bEnable_Shelly9, 
	tDelayRequest:= T#20S, 
	sHostname:= '192.168.178.218', 
	bValidResult=> , 
	bBusy=> , 
	bError=> , 
	bDone=> , 
	hrErrorCode=> ,
	lrPowerTotal=> lrPowerTotal_Shelly9);

// re-calc to kW
lrPowerTotal_Shelly9_kW := lrPowerTotal_Shelly9 / 1000;

(*

// Messung 10
fbShelly10(
	bStart:= bEnable_Shelly10, 
	tDelayRequest:= T#20S, 
	sHostname:= '10.0.0.173', 
	bValidResult=> , 
	bBusy=> , 
	bError=> , 
	bDone=> , 
	hrErrorCode=> ,
	lrPowerTotal=> lrPowerTotal_Shelly10);

// re-calc to kW
lrPowerTotal_Shelly10_kW := lrPowerTotal_Shelly10 / 1000;

// Messung 11
fbShelly11(
	bStart:= bEnable_Shelly11, 
	tDelayRequest:= T#20S, 
	sHostname:= '10.0.0.173', 
	bValidResult=> , 
	bBusy=> , 
	bError=> , 
	bDone=> , 
	hrErrorCode=> ,
	lrPowerTotal=> lrPowerTotal_Shelly11);

// re-calc to kW
lrPowerTotal_Shelly11_kW := lrPowerTotal_Shelly11 / 1000;

// Messung 12
fbShelly12(
	bStart:= bEnable_Shelly12, 
	tDelayRequest:= T#20S, 
	sHostname:= '10.0.0.173', 
	bValidResult=> , 
	bBusy=> , 
	bError=> , 
	bDone=> , 
	hrErrorCode=> ,
	lrPowerTotal=> lrPowerTotal_Shelly12);
	
// re-calc to kW
lrPowerTotal_Shelly12_kW := lrPowerTotal_Shelly12 / 1000;
// sum-up energy
//lrEnergy_M12_Total :=  lrEnergy_M12_L1 + lrEnergy_M12_L2 + lrEnergy_M12_L3;

*)

//other

lrPowerV16_Kitchen_kW := lrPowerTotal_Shelly7_kW + lrPowerTotal_Shelly8_kW + lrPowerTotal_Shelly9_kW;

fbKitchenCounter(
	byActiveTariff:= 1, 
	lrPowerInput:= lrPowerV16_Kitchen_kW, 
	lrTotalCounterEnergy_Consumption=> , 
	lrTotalCounterEnergy_Production=> , 
	lrCounterEnergyT1_Consumption=> , 
	lrCounterEnergyT2_Consumption=> , 
	lrCounterEnergyT1_Production=> , 
	lrCounterEnergyT2_Production=> );
IF fbKitchenCounter.lrTotalCounterEnergy_Consumption > lrPowerV16_Kitchen_kW THEN  	
	lrCounterKitchen := fbKitchenCounter.lrTotalCounterEnergy_Consumption;
END_IF

END_PROGRAM

// ---- FBs/FB_Shelly_Pro3EM.TcPOU
FUNCTION_BLOCK FB_Shelly_Pro3EM
VAR_INPUT
	bStart				: BOOL;
	tDelayRequest		: TIME := T#3S;		//Timer for delay before start with the next read or write Request
	sHostname			: STRING(255);		//Hostname or IP Adress from the Server
END_VAR

VAR_IN_OUT
END_VAR

VAR_OUTPUT
	bValidResult				: BOOL;															//Valid Result received from Server
    bBusy						: BOOL;															//Function is Busy
    bError						: BOOL;															//Error sucess
	bDone						: BOOL;															//True after the decoding from the received Json File
	bConnected					: BOOL;															//Connection to the Server
	lrpowerP1					: LREAL;														//Received Value
	lrfrequencyP1				: LREAL;														//Received Value
	lrcurrentP1					: LREAL;														//Received Value
	lrvoltageP1					: LREAL;														//Received Value
	lrpowerP2					: LREAL;														//Received Value
	lrfrequencyP2				: LREAL;														//Received Value
	lrcurrentP2					: LREAL;														//Received Value
	lrvoltageP2					: LREAL;														//Received Value
	lrpowerP3					: LREAL;														//Received Value
	lrfrequencyP3				: LREAL;														//Received Value
	lrcurrentP3					: LREAL;														//Received Value
	lrvoltageP3					: LREAL;														//Received Value
	lrpowerTotal				: LREAL;														//Received Value
	lrcurrentTotal				: LREAL;														//Received Value
	lrpoweraprtTotal			: LREAL;														//Received Value
	hrErrorCode       			: HRESULT;														//Error Result from Http Client
END_VAR

VAR
	fbClient					: FB_IotHttpClient;
	fbHttpGet					: FB_Shelly_Pro3EM_Helper;
	timStartRequest				: TON;															//Timer to Start the Request
	FPStartRequest				: R_TRIG;														//Internal positive Edge
	FPDone						: R_TRIG;														//Internal positive Edge
	FNStart						: F_TRIG;														//Internal negative Edge
END_VAR

(*------------------------------------------------------------------------------------Configure HTTP Client------------------------------------------------------------------------------------------------------*)

fbClient.sHostName := sHostname;
fbClient.tConnectionTimeout := tDelayRequest;

IF NOT fbClient.bConfigured THEN 
	fbClient.nHostPort:= 80;
	fbClient.bKeepAlive := TRUE;
	fbClient.tConnectionTimeout := T#2S;
END_IF


//Timer to start the Request
FPStartRequest(CLK:= bStart, Q=> );
	timStartRequest(IN:= fbClient.bConfigured AND bStart AND NOT timStartRequest.Q, PT:= tDelayRequest, Q=> , ET=> );
		IF ((timStartRequest.Q AND NOT bBusy) OR (FPStartRequest.Q AND NOT bBusy AND fbClient.bConfigured)) THEN fbHttpGet.bSend := TRUE; END_IF

				
//Http Get Function
fbHttpGet(
	(*lrpowerP1 => lrpowerP1,
	lrfrequencyP1 => lrfrequencyP1,
	lrcurrentP1 => lrcurrentP1,
	lrvoltageP1 => lrvoltageP1,
	lrpowerP2 => lrpowerP2,
	lrfrequencyP2 => lrfrequencyP2,
	lrcurrentP2 => lrcurrentP2,
	lrvoltageP2 => lrvoltageP2,
	lrpowerP3 => lrpowerP3,
	lrfrequencyP3 => lrfrequencyP3,
	lrcurrentP3 => lrcurrentP3,*)
	lr_total_current => lrcurrentTotal,
	lr_total_act_power => lrpowerTotal,
	lr_total_aprt_power => lrpoweraprtTotal,
	bSend:= , 
	fbClient:= fbClient, 
	bBusy=> bBusy, 
	bError=> ,
	sContentS0=> );


fbHttpGet.bSend := FALSE;

FPDone(CLK:= bDone, Q=> );


fbClient.Execute();

//Error
IF fbHttpGet.bError OR fbClient.bError THEN bError := TRUE; ELSE bError := FALSE; END_IF	
	hrErrorCode := fbClient.hrErrorCode;

END_FUNCTION_BLOCK

// ---- FBs/FB_Shelly_Pro3EM_Helper.TcPOU
FUNCTION_BLOCK FB_Shelly_Pro3EM_Helper
VAR_INPUT
	bSend			: BOOL;
END_VAR

VAR_IN_OUT
	fbClient		: FB_IotHttpClient;
END_VAR

VAR_OUTPUT
	bBusy			: BOOL;
	bError			: BOOL;
	
	lr_a_current				: LREAL;	//[A]
	lr_a_voltage				: LREAL;	//[V]
	lr_a_act_power				: LREAL;	//[W]
	lr_a_aprt_power				: LREAL;	//[VA]
	lr_a_pf						: LREAL;	//Phase power factor measurement factor
	lr_a_freq					: LREAL;	//[Hz] 
	
	lr_b_current				: LREAL;	//[A]
	lr_b_voltage				: LREAL;	//[V]
	lr_b_act_power				: LREAL;	//[W]
	lr_b_aprt_power				: LREAL;	//[VA]
	lr_b_pf						: LREAL;	//Phase power factor measurement factor
	lr_b_freq					: LREAL;	//[Hz]
	
	lr_c_current				: LREAL;	//[A]
	lr_c_voltage				: LREAL;	//[V]
	lr_c_act_power				: LREAL;	//[W]
	lr_c_aprt_power				: LREAL;	//[VA]
	lr_c_pf						: LREAL;	//Phase power factor measurement factor
	lr_c_freq					: LREAL;	//[Hz]
	
	lr_total_current			: LREAL;	//[A] 
	lr_total_act_power			: LREAL;	//[W]
	lr_total_aprt_power			: LREAL;	//[VA]
		
	lrpowerP1					: LREAL;
	lrfrequencyP1				: LREAL;
	lrcurrentP1					: LREAL;
	lrvoltageP1					: LREAL;
	lrpowerP2					: LREAL;
	lrfrequencyP2				: LREAL;
	lrcurrentP2					: LREAL;
	lrvoltageP2					: LREAL;
	lrpowerP3					: LREAL;
	lrfrequencyP3				: LREAL;
	lrcurrentP3					: LREAL;
	lrvoltageP3					: LREAL;
	lrpowerTotal				: LREAL;
	lrcurrentTotal				: LREAL;
END_VAR

VAR
	fbRequestStatus		: FB_IotHttpRequest;
	fbJson				: FB_JsonDomParser;
	nState				: UDINT;
	RisingEdge			: R_TRIG;
	timTimeout			: TON;
	tTimeOut			: TIME := T#30S;
	
	bGetContentResult	: BOOL;
	sContentS0			: STRING(8192);
	
	bGetJsonResult		: BOOL;
	jsonDoc				: SJsonValue;
	jsonVal				: SJsonValue;
	
	nReqCount			: UDINT;	
	nResCount			: UDINT;
	nValidResCount		: UDINT;
	nErrCount			: UDINT;
END_VAR

//Timer for Timeout
timTimeout(IN:= nState = 1 AND bBusy, PT:= tTimeOut, Q=> , ET=> );
	IF timTimeout.Q THEN 
		nState := 0;
		bBusy := FALSE;
	END_IF

RisingEdge(CLK:= bSend );
CASE nState OF
0:	
	IF RisingEdge.Q THEN 
		IF fbRequestStatus.SendRequest(sUri:='/rpc/EM.GetStatus?id=0', fbClient:=fbClient, eRequestType:=ETcIotHttpRequestType.HTTP_Get, 0, 0, 0) THEN
			nState:= 1;
			nReqCount:= nReqCount+1;
			bBusy:= TRUE;
			bError:= FALSE;
		END_IF					
	END_IF
1:
	IF NOT fbRequestStatus.bBusy THEN
		bError:= TRUE;
		
		IF NOT fbRequestStatus.bError THEN				 
			bGetContentResult:= fbRequestStatus.GetContent(pContent:= ADR(sContentS0), nContentSize:= SIZEOF(sContentS0), bSetNullTermination:= TRUE);
			IF fbRequestStatus.nStatusCode >= 200 AND fbRequestStatus.nStatusCode < 300 THEN
				bGetJsonResult:= FALSE;
				jsonDoc:= fbRequestStatus.GetJsonDomContent(fbJson);
				IF jsonDoc <> 0 THEN
					bGetJsonResult:= TRUE;
					IF fbJson.HasMember(jsonDoc, 'id')  THEN
						jsonVal:= fbJson.FindMember(jsonDoc, 'a_current');
						nValidResCount:= nValidResCount+1;
						IF fbJson.IsDouble(jsonVal) THEN							
							lr_a_current:= fbJson.GetDouble(jsonVal);									
						END_IF
						jsonVal:= fbJson.FindMember(jsonDoc, 'a_voltage');
						nValidResCount:= nValidResCount+1;					
						IF fbJson.IsDouble(jsonVal) THEN							
							lr_a_voltage:= fbJson.GetDouble(jsonVal);									
						END_IF
						jsonVal:= fbJson.FindMember(jsonDoc, 'a_act_power');
						nValidResCount:= nValidResCount+1;
						IF fbJson.IsDouble(jsonVal) THEN							
							lr_a_act_power:= fbJson.GetDouble(jsonVal);									
						END_IF
						jsonVal:= fbJson.FindMember(jsonDoc, 'a_aprt_power');
						nValidResCount:= nValidResCount+1;
						IF fbJson.IsDouble(jsonVal) THEN							
							lr_a_aprt_power:= fbJson.GetDouble(jsonVal);									
						END_IF
						jsonVal:= fbJson.FindMember(jsonDoc, 'a_pf');
						nValidResCount:= nValidResCount+1;
						IF fbJson.IsDouble(jsonVal) THEN							
							lr_a_pf:= fbJson.GetDouble(jsonVal);									
						END_IF
						jsonVal:= fbJson.FindMember(jsonDoc, 'a_freq');
						nValidResCount:= nValidResCount+1;
						IF fbJson.IsDouble(jsonVal) THEN							
							lr_a_freq:= fbJson.GetDouble(jsonVal);									
						END_IF
						bError:= FALSE;
					END_IF						
				nResCount:= nResCount+1;			
				END_IF
			END_IF
		END_IF
		
		IF NOT fbRequestStatus.bError THEN				 
			bGetContentResult:= fbRequestStatus.GetContent(pContent:= ADR(sContentS0), nContentSize:= SIZEOF(sContentS0), bSetNullTermination:= TRUE);
			IF fbRequestStatus.nStatusCode >= 200 AND fbRequestStatus.nStatusCode < 300 THEN
				bGetJsonResult:= FALSE;
				jsonDoc:= fbRequestStatus.GetJsonDomContent(fbJson);
				IF jsonDoc <> 0 THEN
					bGetJsonResult:= TRUE;
					IF fbJson.HasMember(jsonDoc, 'id')  THEN
						jsonVal:= fbJson.FindMember(jsonDoc, 'b_current');
						nValidResCount:= nValidResCount+1;
						IF fbJson.IsDouble(jsonVal) THEN							
							lr_b_current:= fbJson.GetDouble(jsonVal);									
						END_IF
						jsonVal:= fbJson.FindMember(jsonDoc, 'b_voltage');
						nValidResCount:= nValidResCount+1;					
						IF fbJson.IsDouble(jsonVal) THEN							
							lr_b_voltage:= fbJson.GetDouble(jsonVal);									
						END_IF
						jsonVal:= fbJson.FindMember(jsonDoc, 'b_act_power');
						nValidResCount:= nValidResCount+1;
						IF fbJson.IsDouble(jsonVal) THEN							
							lr_b_act_power:= fbJson.GetDouble(jsonVal);									
						END_IF
						jsonVal:= fbJson.FindMember(jsonDoc, 'b_aprt_power');
						nValidResCount:= nValidResCount+1;
						IF fbJson.IsDouble(jsonVal) THEN							
							lr_b_aprt_power:= fbJson.GetDouble(jsonVal);									
						END_IF
						jsonVal:= fbJson.FindMember(jsonDoc, 'b_pf');
						nValidResCount:= nValidResCount+1;
						IF fbJson.IsDouble(jsonVal) THEN							
							lr_b_pf:= fbJson.GetDouble(jsonVal);									
						END_IF
						jsonVal:= fbJson.FindMember(jsonDoc, 'b_freq');
						nValidResCount:= nValidResCount+1;
						IF fbJson.IsDouble(jsonVal) THEN							
							lr_b_freq:= fbJson.GetDouble(jsonVal);									
						END_IF
						bError:= FALSE;
					END_IF						
				nResCount:= nResCount+1;			
				END_IF
			END_IF
		END_IF
		
		IF NOT fbRequestStatus.bError THEN				 
			bGetContentResult:= fbRequestStatus.GetContent(pContent:= ADR(sContentS0), nContentSize:= SIZEOF(sContentS0), bSetNullTermination:= TRUE);
			IF fbRequestStatus.nStatusCode >= 200 AND fbRequestStatus.nStatusCode < 300 THEN
				bGetJsonResult:= FALSE;
				jsonDoc:= fbRequestStatus.GetJsonDomContent(fbJson);
				IF jsonDoc <> 0 THEN
					bGetJsonResult:= TRUE;
					IF fbJson.HasMember(jsonDoc, 'id')  THEN
						jsonVal:= fbJson.FindMember(jsonDoc, 'c_current');
						nValidResCount:= nValidResCount+1;
						IF fbJson.IsDouble(jsonVal) THEN							
							lr_c_current:= fbJson.GetDouble(jsonVal);									
						END_IF
						jsonVal:= fbJson.FindMember(jsonDoc, 'c_voltage');
						nValidResCount:= nValidResCount+1;					
						IF fbJson.IsDouble(jsonVal) THEN							
							lr_c_voltage:= fbJson.GetDouble(jsonVal);									
						END_IF
						jsonVal:= fbJson.FindMember(jsonDoc, 'c_act_power');
						nValidResCount:= nValidResCount+1;
						IF fbJson.IsDouble(jsonVal) THEN							
							lr_c_act_power:= fbJson.GetDouble(jsonVal);									
						END_IF
						jsonVal:= fbJson.FindMember(jsonDoc, 'c_aprt_power');
						nValidResCount:= nValidResCount+1;
						IF fbJson.IsDouble(jsonVal) THEN							
							lr_c_aprt_power:= fbJson.GetDouble(jsonVal);									
						END_IF
						jsonVal:= fbJson.FindMember(jsonDoc, 'c_pf');
						nValidResCount:= nValidResCount+1;
						IF fbJson.IsDouble(jsonVal) THEN							
							lr_c_pf:= fbJson.GetDouble(jsonVal);									
						END_IF
						jsonVal:= fbJson.FindMember(jsonDoc, 'c_freq');
						nValidResCount:= nValidResCount+1;
						IF fbJson.IsDouble(jsonVal) THEN							
							lr_c_freq:= fbJson.GetDouble(jsonVal);									
						END_IF
						bError:= FALSE;
					END_IF						
				nResCount:= nResCount+1;			
				END_IF
			END_IF
		END_IF
		
		IF NOT fbRequestStatus.bError THEN				 
			bGetContentResult:= fbRequestStatus.GetContent(pContent:= ADR(sContentS0), nContentSize:= SIZEOF(sContentS0), bSetNullTermination:= TRUE);
			IF fbRequestStatus.nStatusCode >= 200 AND fbRequestStatus.nStatusCode < 300 THEN
				bGetJsonResult:= FALSE;
				jsonDoc:= fbRequestStatus.GetJsonDomContent(fbJson);
				IF jsonDoc <> 0 THEN
					bGetJsonResult:= TRUE;
                        IF fbJson.HasMember(jsonDoc, 'id') THEN
                            jsonVal:= fbJson.FindMember(jsonDoc, 'total_current');
                            nValidResCount:= nValidResCount+1;
                            IF fbJson.IsDouble(jsonVal) THEN
                                lr_total_current:= fbJson.GetDouble(jsonVal);
                            END_IF
							jsonVal:= fbJson.FindMember(jsonDoc, 'total_act_power');
                            nValidResCount:= nValidResCount+1;
                            IF fbJson.IsDouble(jsonVal) THEN
                                lr_total_act_power:= fbJson.GetDouble(jsonVal);
                            END_IF
							jsonVal:= fbJson.FindMember(jsonDoc, 'total_aprt_power');
                            nValidResCount:= nValidResCount+1;
                            IF fbJson.IsDouble(jsonVal) THEN
                                lr_total_aprt_power:= fbJson.GetDouble(jsonVal);
                            END_IF
						bError:= FALSE;
						END_IF					
				nResCount:= nResCount+1;			
				END_IF
			END_IF
		END_IF
		(*
		IF NOT fbRequestSwitch1.bError THEN				 
			bGetContentResult:= fbRequestSwitch1.GetContent(pContent:= ADR(sContentS1), nContentSize:= SIZEOF(sContentS1), bSetNullTermination:= TRUE);
			IF fbRequestSwitch1.nStatusCode >= 200 AND fbRequestSwitch1.nStatusCode < 300 THEN
				bGetJsonResult:= FALSE;
				jsonDoc:= fbRequestSwitch1.GetJsonDomContent(fbJson);
				IF jsonDoc <> 0 THEN
					bGetJsonResult:= TRUE;
					IF fbJson.HasMember(jsonDoc, 'output')  THEN
                        IF fbJson.HasMember(jsonVal, 'total') THEN
                            jsonVal:= fbJson.FindMember(jsonVal, 'total');
                            nValidResCount:= nValidResCount+1;
                            IF fbJson.IsDouble(jsonVal) THEN
                                lraenergyP2:= fbJson.GetDouble(jsonVal);
                            END_IF
						bError:= FALSE;
						END_IF
					END_IF						
				nResCount:= nResCount+1;			
				END_IF
			END_IF
		END_IF
		
		IF NOT fbRequestSwitch2.bError THEN				 
			bGetContentResult:= fbRequestSwitch2.GetContent(pContent:= ADR(sContentS2), nContentSize:= SIZEOF(sContentS2), bSetNullTermination:= TRUE);
			IF fbRequestSwitch2.nStatusCode >= 200 AND fbRequestSwitch2.nStatusCode < 300 THEN
				bGetJsonResult:= FALSE;
				jsonDoc:= fbRequestSwitch2.GetJsonDomContent(fbJson);
				IF jsonDoc <> 0 THEN
					bGetJsonResult:= TRUE;
					IF fbJson.HasMember(jsonDoc, 'output')  THEN
						jsonVal:= fbJson.FindMember(jsonDoc, 'apower');
						nValidResCount:= nValidResCount+1;
						IF fbJson.IsDouble(jsonVal) THEN							
							lrapowerP3:= fbJson.GetDouble(jsonVal);									
						END_IF
						jsonVal:= fbJson.FindMember(jsonDoc, 'voltage');
						nValidResCount:= nValidResCount+1;					
						IF fbJson.IsDouble(jsonVal) THEN							
							lrvoltageP3:= fbJson.GetDouble(jsonVal);									
						END_IF
						jsonVal:= fbJson.FindMember(jsonDoc, 'aenergy');
                        IF fbJson.HasMember(jsonVal, 'total') THEN
                            jsonVal:= fbJson.FindMember(jsonVal, 'total');
                            nValidResCount:= nValidResCount+1;
                            IF fbJson.IsDouble(jsonVal) THEN
                                lraenergyP3:= fbJson.GetDouble(jsonVal);
                            END_IF
						bError:= FALSE;
						END_IF
					END_IF						
				nResCount:= nResCount+1;			
				END_IF
			END_IF
		END_IF
		
		IF NOT fbRequestSwitch3.bError THEN				 
			bGetContentResult:= fbRequestSwitch3.GetContent(pContent:= ADR(sContentS3), nContentSize:= SIZEOF(sContentS3), bSetNullTermination:= TRUE);
			IF fbRequestSwitch3.nStatusCode >= 200 AND fbRequestSwitch3.nStatusCode < 300 THEN
				bGetJsonResult:= FALSE;
				jsonDoc:= fbRequestSwitch3.GetJsonDomContent(fbJson);
				IF jsonDoc <> 0 THEN
					bGetJsonResult:= TRUE;
					IF fbJson.HasMember(jsonDoc, 'output')  THEN
						jsonVal:= fbJson.FindMember(jsonDoc, 'apower');
						nValidResCount:= nValidResCount+1;
						IF fbJson.IsDouble(jsonVal) THEN							
							lrapowerP4:= fbJson.GetDouble(jsonVal);									
						END_IF
						jsonVal:= fbJson.FindMember(jsonDoc, 'voltage');
						nValidResCount:= nValidResCount+1;					
						IF fbJson.IsDouble(jsonVal) THEN							
							lrvoltageP4:= fbJson.GetDouble(jsonVal);									
						END_IF
						jsonVal:= fbJson.FindMember(jsonDoc, 'aenergy');
                        IF fbJson.HasMember(jsonVal, 'total') THEN
                            jsonVal:= fbJson.FindMember(jsonVal, 'total');
                            nValidResCount:= nValidResCount+1;
                            IF fbJson.IsDouble(jsonVal) THEN
                                lraenergyP4:= fbJson.GetDouble(jsonVal);
                            END_IF
						bError:= FALSE;
						END_IF
					END_IF						
				nResCount:= nResCount+1;			
				END_IF
			END_IF
		END_IF
		*)
	nState:= 0;
	bBusy:= FALSE;
		IF bError THEN
			nErrCount:= nErrCount+1;
		END_IF
	END_IF  	
END_CASE

fbClient.Execute();

END_FUNCTION_BLOCK

// ---- POUs/prgComEffIO.TcPOU
PROGRAM prgComEffIO
VAR
	fbCom					: FB_MqttCommunicator_V2;
	stringArray_Last_HB		: ARRAY[0..50] OF STRING(30);
END_VAR

fbCom(
	bConnect:= TRUE, 
	strAuthKey:=  'BE736352867778' ,
	sUserName:= 'bd8cddef-7a46-4cb7-9100-c3c67f8ed94a', 
	sUserPassword:= '26bcb4df-2135-49e0-bf55-9c706b8073f9', 
	eSavePositionCertificate:= eSavePositionOnPLC.ePostionHardDisk, 
	bConnected=> , 
	bError=> , 
	hrErrorCode=> , 
	eConnectionState=> , 
	eErrorMessage_Out=> );

END_PROGRAM

// ---- FBs/FB_MqttCommunicator_V2_1.TcPOU
{attribute 'hide_all_locals'}
FUNCTION_BLOCK FB_MqttCommunicator_V2_1
VAR_INPUT
	bConnect      				: BOOL;															//If True then a connection to the cloud service is established
	strAuthKey					: String (20);													//Customer Authentication Key, provided from EfficientIO
	sUserName     				: STRING(36);     												//Username that was given in the cloud when the project was created
    sUserPassword 				: STRING(36);   					 							//Password that was given in the cloud when the project was created
	eSavePositionCertificate	: eSavePositionOnPLC;											//Save Position from the certificate (HardDisk\ or C:\) 
	time_HeartBeat_sec			: TIME:=T#60S;													// Heart Beat Time 					
END_VAR
VAR_OUTPUT
	bConnected					: BOOL;															//True = PLC is Connected to the cloud service FALSE = Not connected
	bError          			: BOOL;															//Error flag
    hrErrorCode      			: HRESULT;														//Error code if bError is true
    eConnectionState 			: ETcIotMqttClientState;										//State of the cloud connection
	eErrorMessage_Out			: eErrorMessage;												//Error State from received Messege
END_VAR
VAR
	(*-----------------------------------------------------Other-----------------------------------------------------------------------------------------*)
	fbMqttClient    			: FB_IotMqttClient;												//Function mqtt client
	fbJsonWrite					: FB_MessageWrite;												//Json Write function
	fbJsonRead					: FB_MessageRead;												//Json Read function
	fbGetTime					: NT_GetTime;													//System time
	FNGetTimeDate				: F_TRIG;														//Intern falling edge
	timError					: TON;															//Timer error to clear Message Queue
    bSetParameter   			: BOOL := TRUE;													//Set new parameter
	bClientIDCreated			: BOOL;															//True if the client id is generated
	byLPCopyValuesGV_1			: BYTE;															//Loop to copy the data from global interface in the read Json function
	udiLPCopyValuesGV_2			: UDINT;														//Loop to copy the data from global interface in the read Json function
	sUserNameOld     			: STRING(36);    												//Old User name from the project
    sUserPasswordOld 			: STRING(36);    												//Old Password for the project
	sClientID					: STRING(255);													//Client ID
	eSavePositionCertificateOld	: eSavePositionOnPLC;											//Old Position from the certificate (HardDisk\ or C:\) 
	(*---------------------------------------------------published message---------------------------------------------------------------------------*)
	arrBusySendigInterface		: ARRAY[1..10] OF BOOL;											//Array to save with what Send Interface it was sending the last message to enbale that after sending for new Message
	arrTimoutSendinigInterface	: ARRAY[1..10] OF TON;											//Timer to Reset a Sending Interface after a Delay. That its not possible to block everytime the sending interface 
   	bHBSending					: BOOL;															//Heart Beat Sending is in progress
	byLPJsonSend				: BYTE;															//Loop to prepear data befor sending
	byLPSendInterface			: BYTE;															//Loop for the send interface
	uiStatePublish				: UINT;															//State maschine sending
	sTopicPub   				: STRING(255);													//Topic publish
    sPayloadPub 				: STRING(7000);													//Payload publish
    fbTimerPub 					: TON;															//Timer to send the message to the broker after expiration of time 
	fbTimerHB					: TON;															//Timer for sending the Heart Beat
	(*---------------------------------------------------received message----------------------------------------------------------------------------*)
    bSubscribed    				: BOOL;															//True if the connection to the broker is on
	bUnsubscribe				: BOOL;															//True if the connection to the broker is off
	bReadOut					: BOOL;															//Read out value from received buffer
	bBusyWrite					: BOOL;															//Interface write is busy	
	bErrorWrite					: BOOL;															//Interface write has a error
	byCounterBusyErrorWrite		: BYTE;															//Counter to clear error or busy state
    byLPWriteInterface			: BYTE;															//Loop for the write interface
	sTopicSub      				: STRING(255);													//Topic subscrib
	{attribute 'TcEncoding':='UTF-8'}
  	sPayloadRcv    				: STRING(7000);													//Payload received
  	fbMessageQueue 				: FB_IotMqttMessageQueue;										//Function message queuee
    fbMessage      				: FB_IotMqttMessage;											//Function message
	int_Target: INT;
	str_sHostName				: STRING(40);
	str_Certificate				: STRING(100);
END_VAR

//Creator : Stefan Lackner
//Company : EfficientIO
//Date : 06.12.2022
//Version : 2.1

//With this function we can commiunicate over mqtt with the ventus cloud service to write data from plc to the cloud or receive data from cloud and write to plc
//Max data from cloud to the plc is every 250MS 1 messege.
//Data from plc to cloud is every 50MS if messages are in the buffer from the interface
//So that the mqtt function starts, the scann function must be completed  

// SL: V2: Added input time_HeartBeat_sec for adjustable heart beat
// SL  V2.1: Added input strAuthKey with related IF (LIne 25-54. Changed str_sHostName and str_Certificate accordingly. 

//Create Client ID
fbGetTime(START:= NOT bClientIDCreated,);
	FNGetTimeDate(CLK:= fbGetTime.BUSY, Q=> );

IF FNGetTimeDate.Q AND NOT fbGetTime.ERR THEN
	sClientID := CONCAT(CONCAT(WORD_TO_STRING(fbGetTime.TIMESTR.wYear),WORD_TO_STRING(fbGetTime.TIMESTR.wMonth)),CONCAT(CONCAT(WORD_TO_STRING(fbGetTime.TIMESTR.wDay),WORD_TO_STRING(fbGetTime.TIMESTR.wDayOfWeek)),CONCAT(CONCAT(WORD_TO_STRING(fbGetTime.TIMESTR.wHour),WORD_TO_STRING(fbGetTime.TIMESTR.wMinute)),
					CONCAT(CONCAT(WORD_TO_STRING(fbGetTime.TIMESTR.wSecond),WORD_TO_STRING(fbGetTime.TIMESTR.wMilliseconds)),TwinCAT_SystemInfoVarList._AppInfo.ProjectName))));
		bClientIDCreated := TRUE;
END_IF		


// find out which designation String is selected
IF strAuthKey = 'EIO08031879806' THEN			// EfficientIO
	str_sHostName	:= 'mqtt.efficientio.com';
	IF eSavePositionCertificate = eSavePositionOnPLC.ePostionHardDisk THEN 
		str_Certificate      := 'Hard Disk\TwinCAT\3.1\Config\Certificates\mqtt.pem';
	ELSIF eSavePositionCertificate = eSavePositionOnPLC.ePostionC THEN
		str_Certificate      := 'C:\TwinCAT\3.1\Config\Certificates\mqtt.pem';		
	END_IF	
ELSIF strAuthKey = 'TSG88376368072' THEN		// TSG
	str_sHostName	:= 'mqtt.tsg-portal.de';
	IF eSavePositionCertificate = eSavePositionOnPLC.ePostionHardDisk THEN 
		str_Certificate      := 'Hard Disk\TwinCAT\3.1\Config\Certificates\mqtt_tsg.pem';
	ELSIF eSavePositionCertificate = eSavePositionOnPLC.ePostionC THEN
		str_Certificate      := 'C:\TwinCAT\3.1\Config\Certificates\mqtt_tsg.pem';	
	END_IF	
ELSIF strAuthKey = 'BE736352867778' THEN		//Burgenland Energie
	str_sHostName	:= 'mqtt.leo-b2b.burgenlandenergie.at';
	IF eSavePositionCertificate = eSavePositionOnPLC.ePostionHardDisk THEN 
		str_Certificate      := 'Hard Disk\TwinCAT\3.1\Config\Certificates\mqtt_be.pem';
	ELSIF eSavePositionCertificate = eSavePositionOnPLC.ePostionC THEN
		str_Certificate      := 'C:\TwinCAT\3.1\Config\Certificates\mqtt_be.pem';	
	END_IF	
ELSIF strAuthKey = 'PEN94103490274' THEN		//Peneder
	str_sHostName	:= 'mqtt.connect.peneder.com';
	IF eSavePositionCertificate = eSavePositionOnPLC.ePostionHardDisk THEN 
		str_Certificate      := 'Hard Disk\TwinCAT\3.1\Config\Certificates\mqtt_peneder.pem';
	ELSIF eSavePositionCertificate = eSavePositionOnPLC.ePostionC THEN
		str_Certificate      := 'C:\TwinCAT\3.1\Config\Certificates\mqtt_peneder.pem';	
	END_IF	
END_IF

IF bSetParameter AND bClientIDCreated THEN
    bSetParameter               := FALSE;
	fbMqttClient.sClientId		:= sClientID;
    fbMqttClient.sHostName      := str_sHostName;
    fbMqttClient.nHostPort      := 8883;
  	fbMqttClient.sTopicPrefix   := ''; 
	fbMqttClient.nKeepAlive     := 30; 
	fbMqttClient.sUserName      := sUserName;
	fbMqttClient.sUserPassword  := sUserPassword; 
	//TLS
	fbMqttClient.stTLS.sCA      := str_Certificate;

	fbMqttClient.stTLS.sVersion	:= 'tlsv1.2';
    fbMqttClient.ipMessageQueue := fbMessageQueue;
END_IF

//Config timer pub
fbTimerPub.PT := T#25MS;

//Change Inputs and disconnect connection
IF sUserName <> sUserNameOld OR sUserPassword <> sUserPasswordOld OR eSavePositionCertificate <> eSavePositionCertificateOld THEN 
	bConnect := FALSE; bSetParameter := TRUE; sUserNameOld := sUserName; sUserPasswordOld := sUserPassword; 
		eSavePositionCertificateOld := eSavePositionCertificate;	
END_IF 

//Subscribe and Unsubscribe befor remove client connection
IF NOT bConnect OR Lynus_Standards.GVL_Communicator.bBusyInfoAlVariables OR Lynus_Standards.GVL_Communicator.bErrorInfoAlVariables OR NOT Lynus_Standards.GVL_Communicator.bInfoAlVariablesOK THEN
	IF NOT bUnsubscribe THEN
		bUnsubscribe := fbMqttClient.Unsubscribe(sTopic:= sTopicSub);
	END_IF
		fbMqttClient.Execute(FALSE);
			bSubscribed := FALSE;
				//Stop ADS read/write when the connection to the broker is off and clear the received buffer
				FOR byLPSendInterface := 1 TO 10 BY 1 DO 
					Lynus_Standards.GVL_Communicator.arrInterfaceInfoValueSendTo[byLPSendInterface].bBusy := FALSE;
						Lynus_Standards.GVL_Communicator.arrInterfaceInfoValueSendTo[byLPSendInterface].bErrorSending := TRUE;
							arrBusySendigInterface[byLPSendInterface] := FALSE;
				END_FOR
					fbTimerPub(IN:= FALSE); bReadOut := FALSE; 	bBusyWrite := FALSE; bErrorWrite := FALSE;
						sPayloadRcv := ''; uiStatePublish := 0;
							fbMessageQueue.ResetQueue();										
ELSE
	IF NOT bSetParameter AND NOT Lynus_Standards.GVL_Communicator.bBusyInfoAlVariables AND NOT Lynus_Standards.GVL_Communicator.bErrorInfoAlVariables AND Lynus_Standards.GVL_Communicator.bInfoAlVariablesOK THEN
		bUnsubscribe := FALSE;
			fbMqttClient.Execute(TRUE);
				//Start ADS read/write when the connection to the broker is on and no error
				IF NOT fbMqttClient.bError AND fbMqttClient.bConnected THEN 
					FOR byLPSendInterface := 1 TO 10 BY 1 DO 
						Lynus_Standards.GVL_Communicator.arrInterfaceInfoValueSendTo[byLPSendInterface].bErrorSending := FALSE;
					END_FOR
				ELSE 
					//Stop read/write and clear the received buffer from old messages
					FOR byLPSendInterface := 1 TO 10 BY 1 DO 
						Lynus_Standards.GVL_Communicator.arrInterfaceInfoValueSendTo[byLPSendInterface].bErrorSending := TRUE;
							arrBusySendigInterface[byLPSendInterface] := FALSE;
					END_FOR
						bReadOut := FALSE; bBusyWrite := FALSE; bErrorWrite := FALSE;
							sPayloadRcv := ''; uiStatePublish := 0;
								fbMessageQueue.ResetQueue();
				END_IF		
	END_IF	
END_IF

(*----------------------------------------------------------------------------------Send Messeges---------------------------------------------------------------*)

//Prepare Json Doc for sending
time_HeartBeat_sec := LIMIT (T#5S,time_HeartBeat_sec,T#3600S);
IF bConnected AND NOT bError AND NOT bHBSending THEN fbTimerHB.IN := TRUE; ELSE fbTimerHB.IN := FALSE; END_IF
	fbTimerHB(IN:= , PT:= time_HeartBeat_sec, Q=> , ET=> );

IF Lynus_Standards.GVL_Communicator.byNumberOfReadWriteFunction >= 1 AND Lynus_Standards.GVL_Communicator.byNumberOfReadWriteFunction <= 10 THEN	
	FOR byLPJsonSend := 1 TO Lynus_Standards.GVL_Communicator.byNumberOfReadWriteFunction BY 1 DO 	
		fbJsonWrite.stInfoToConvertInMessage[byLPJsonSend].sFullSymbolName := Lynus_Standards.GVL_Communicator.arrInterfaceInfoValueSendTo[byLPJsonSend].sFullSymbolName;
			fbJsonWrite.stInfoToConvertInMessage[byLPJsonSend].sSymbolUnit := Lynus_Standards.GVL_Communicator.arrInterfaceInfoValueSendTo[byLPJsonSend].sSymbolUnit; 
				fbJsonWrite.stInfoToConvertInMessage[byLPJsonSend].sSymbolType := Lynus_Standards.GVL_Communicator.arrInterfaceInfoValueSendTo[byLPJsonSend].sSymbolType;
					fbJsonWrite.stInfoToConvertInMessage[byLPJsonSend].arrValue := Lynus_Standards.GVL_Communicator.arrInterfaceInfoValueSendTo[byLPJsonSend].arrValue; 	
	END_FOR 	
END_IF

//Heart Beat			
IF (fbTimerHB.Q AND uiStatePublish = 0) OR bHBSending THEN
	fbJsonWrite.stInfoToConvertInMessage[1].sFullSymbolName := '';
		fbJsonWrite.stInfoToConvertInMessage[1].sSymbolUnit := ''; 
			fbJsonWrite.stInfoToConvertInMessage[1].sSymbolType := 'STRING(30)';
				fbJsonWrite.stInfoToConvertInMessage[1].arrValue[1] := 'hb';
					bHBSending := TRUE;
	FOR byLPJsonSend := 2 TO 10 BY 1 DO
		fbJsonWrite.stInfoToConvertInMessage[byLPJsonSend].sFullSymbolName := '';
			fbJsonWrite.stInfoToConvertInMessage[byLPJsonSend].sSymbolUnit := ''; 
				fbJsonWrite.stInfoToConvertInMessage[byLPJsonSend].sSymbolType := '';
					fbJsonWrite.stInfoToConvertInMessage[byLPJsonSend].arrValue[1] := '';
	END_FOR
END_IF  			

IF uiStatePublish = 0 THEN fbJsonWrite.bEnable := TRUE; END_IF
			
fbJsonWrite(stInfoToConvertInMessage:= , sMessageDocToWrite=> sPayloadPub, eErrorMessage_Out => ,);

//Publish
IF fbMqttClient.bConnected AND NOT bSetParameter THEN
    IF NOT bSubscribed THEN
        bSubscribed := fbMqttClient.Subscribe(sTopic:= sTopicSub, eQoS:=TcIotMqttQos.AtMostOnceDelivery);
    END_IF
 END_IF

//Topics
sTopicPub := CONCAT(CONCAT('projects/',sUserName),'/messages');
	sTopicSub := CONCAT(CONCAT('projects/',sUserName),'/messages2'); 
 
CASE uiStatePublish OF
	
	0://Wait to publish
		IF NOT bHBSending THEN
			IF Lynus_Standards.GVL_Communicator.byNumberOfReadWriteFunction >= 1 AND Lynus_Standards.GVL_Communicator.byNumberOfReadWriteFunction <= 10 THEN
				FOR byLPJsonSend := 1 TO Lynus_Standards.GVL_Communicator.byNumberOfReadWriteFunction BY 1 DO
					IF Lynus_Standards.GVL_Communicator.arrInterfaceInfoValueSendTo[byLPJsonSend].bBusy AND fbJsonWrite.bDone THEN 
						uiStatePublish := 1; 
							arrBusySendigInterface[byLPJsonSend] := TRUE;
								fbJsonWrite.bEnable := FALSE;
					END_IF
				END_FOR
			END_IF
		END_IF
			IF bHBSending AND fbJsonWrite.bDone THEN uiStatePublish := 2; fbJsonWrite.bEnable := FALSE; END_IF
			
	1://Publish the message
		fbTimerPub(IN := TRUE);
			IF fbTimerPub.Q THEN // publish new payload every 25MS if messages are in the buffer after ads read
				fbTimerPub(IN := FALSE);
					IF Lynus_Standards.GVL_Communicator.byNumberOfReadWriteFunction >= 1 AND Lynus_Standards.GVL_Communicator.byNumberOfReadWriteFunction <= 10 THEN
						FOR byLPJsonSend := 1 TO Lynus_Standards.GVL_Communicator.byNumberOfReadWriteFunction BY 1 DO
							//Mark the sendet variables on interfaces as done
							IF arrBusySendigInterface[byLPJsonSend] THEN 
								Lynus_Standards.GVL_Communicator.arrInterfaceInfoValueSendTo[byLPJsonSend].bBusy := FALSE; 
									arrBusySendigInterface[byLPJsonSend] := FALSE; 
										Lynus_Standards.GVL_Communicator.arrInterfaceInfoValueSendTo[byLPJsonSend].sSymbolType := '';	
							END_IF
						END_FOR
					END_IF
						IF NOT fbJsonWrite.bError THEN 
							fbMqttClient.Publish(sTopic:= sTopicPub, 
													pPayload:= ADR(sPayloadPub), nPayloadSize:= LEN2(ADR(sPayloadPub)), 
													eQoS:= TcIotMqttQos.AtMostOnceDelivery, bRetain:= FALSE, bQueue:= FALSE);	
						END_IF
													uiStatePublish := 0;
			END_IF	
		
	2://Publish the HB Message
		IF NOT fbJsonWrite.bError THEN
			fbMqttClient.Publish(sTopic:= sTopicPub, 
									pPayload:= ADR(sPayloadPub), nPayloadSize:= LEN2(ADR(sPayloadPub)), 
									eQoS:= TcIotMqttQos.AtMostOnceDelivery, bRetain:= FALSE, bQueue:= FALSE);
		END_IF
								
			bHBSending := FALSE;					
				uiStatePublish := 0;

END_CASE

//Reset the Sending Interface after it is to long time busy to enable it for a new Messages from the Buffer
FOR byLPJsonSend := 1 TO 10 BY 1 DO
	IF Lynus_Standards.GVL_Communicator.arrInterfaceInfoValueSendTo[byLPJsonSend].bBusy THEN arrTimoutSendinigInterface[byLPJsonSend].IN := TRUE; ELSE arrTimoutSendinigInterface[byLPJsonSend].IN := FALSE; END_IF
		IF arrTimoutSendinigInterface[byLPJsonSend].Q THEN 
			Lynus_Standards.GVL_Communicator.arrInterfaceInfoValueSendTo[byLPJsonSend].bBusy := FALSE;
				arrBusySendigInterface[byLPJsonSend] := FALSE;
					Lynus_Standards.GVL_Communicator.arrInterfaceInfoValueSendTo[byLPJsonSend].sSymbolType := '';	
		END_IF    
END_FOR

arrTimoutSendinigInterface[1](IN:= , PT:= T#15S, Q=> , ET=> );
arrTimoutSendinigInterface[2](IN:= , PT:= T#15S, Q=> , ET=> );
arrTimoutSendinigInterface[3](IN:= , PT:= T#15S, Q=> , ET=> );
arrTimoutSendinigInterface[4](IN:= , PT:= T#15S, Q=> , ET=> );
arrTimoutSendinigInterface[5](IN:= , PT:= T#15S, Q=> , ET=> );
arrTimoutSendinigInterface[6](IN:= , PT:= T#15S, Q=> , ET=> );
arrTimoutSendinigInterface[7](IN:= , PT:= T#15S, Q=> , ET=> );
arrTimoutSendinigInterface[8](IN:= , PT:= T#15S, Q=> , ET=> );
arrTimoutSendinigInterface[9](IN:= , PT:= T#15S, Q=> , ET=> );
arrTimoutSendinigInterface[10](IN:= , PT:= T#15S, Q=> , ET=> );

(*----------------------------------------------------------------------------------Received Messeges---------------------------------------------------------------*)

byCounterBusyErrorWrite := 0;

//Busy write interface
IF Lynus_Standards.GVL_Communicator.byNumberOfReadWriteFunction >= 1 AND Lynus_Standards.GVL_Communicator.byNumberOfReadWriteFunction <= 10 THEN 
	FOR byLPWriteInterface := 1 TO Lynus_Standards.GVL_Communicator.byNumberOfReadWriteFunction BY 1 DO 
		IF Lynus_Standards.GVL_Communicator.arrInterfaceInfoValueWriteTo[byLPWriteInterface].bBusy THEN bBusyWrite := TRUE; END_IF
		IF NOT Lynus_Standards.GVL_Communicator.arrInterfaceInfoValueWriteTo[byLPWriteInterface].bBusy THEN byCounterBusyErrorWrite := byCounterBusyErrorWrite + 1; END_IF  
	END_FOR 
END_IF
	IF byCounterBusyErrorWrite >= Lynus_Standards.GVL_Communicator.byNumberOfReadWriteFunction THEN bBusyWrite := FALSE; END_IF

byCounterBusyErrorWrite := 0;

//Error on a write interface
IF Lynus_Standards.GVL_Communicator.byNumberOfReadWriteFunction >= 1 AND Lynus_Standards.GVL_Communicator.byNumberOfReadWriteFunction <= 10 THEN 
	FOR byLPWriteInterface := 1 TO Lynus_Standards.GVL_Communicator.byNumberOfReadWriteFunction BY 1 DO 
		IF Lynus_Standards.GVL_Communicator.arrInterfaceInfoValueWriteTo[byLPWriteInterface].bErrorWrite THEN bErrorWrite := TRUE; END_IF
		IF NOT Lynus_Standards.GVL_Communicator.arrInterfaceInfoValueWriteTo[byLPWriteInterface].bErrorWrite THEN byCounterBusyErrorWrite := byCounterBusyErrorWrite + 1; END_IF  
	END_FOR 
END_IF
	IF byCounterBusyErrorWrite >= Lynus_Standards.GVL_Communicator.byNumberOfReadWriteFunction THEN bErrorWrite := FALSE; END_IF 
	 
IF fbMqttClient.bConnected AND NOT fbMqttClient.bError AND NOT bBusyWrite AND NOT bErrorWrite THEN bReadOut := TRUE; ELSE bReadOut := FALSE; END_IF  

IF (fbMessageQueue.nQueuedMessages > 0 AND bReadOut) OR
	(fbMessageQueue.nQueuedMessages > 0 AND bReadOut AND (fbJsonRead.bError)) THEN
		IF fbMessageQueue.Dequeue(fbMessage:=fbMessage) THEN
			IF fbMessage.CompareTopic(sTopicSub) THEN
				fbMessage.GetPayload(pPayload:=ADR(sPayloadRcv), nPayloadSize:=SIZEOF(sPayloadRcv), bSetNullTermination:= TRUE);
			END_IF
		END_IF
END_IF

//Copy only as much data as you have to save resources
IF Lynus_Standards.GVL_Communicator.byNumberOfReadWriteFunction >= 1 AND Lynus_Standards.GVL_Communicator.byNumberOfReadWriteFunction <= 10 THEN
	FOR byLPCopyValuesGV_1 := 1 TO Lynus_Standards.GVL_Communicator.byNumberOfReadWriteFunction BY 1 DO
		IF Lynus_Standards.GVL_Communicator.arrCounterVariableInArray[byLPCopyValuesGV_1] >= 1 AND Lynus_Standards.GVL_Communicator.arrCounterVariableInArray[byLPCopyValuesGV_1] <= Lynus_Standards.Constants_Communicator.udiArraySizeMarkedSymobls THEN
			FOR udiLPCopyValuesGV_2 := 1 TO Lynus_Standards.GVL_Communicator.arrCounterVariableInArray[byLPCopyValuesGV_1] BY 1 DO  			
				fbJsonRead.arrVarInfos[byLPCopyValuesGV_1,udiLPCopyValuesGV_2] := Lynus_Standards.GVL_Communicator.arrInterfaceInfoAlVariables[byLPCopyValuesGV_1,udiLPCopyValuesGV_2];	
			END_FOR
		END_IF 
	END_FOR
END_IF    

fbJsonRead(
	sReceivedMessageDoc:= sPayloadRcv, 
	arrVarInfos:= , 
	stInfoFromReceivedMessage=> , 
	bError=> , 
	bMuchMoreInformationReceived=> , 
	eErrorMessage_Out=> );

IF NOT fbJsonRead.bError AND bReadOut AND fbJsonRead.stInfoFromReceivedMessage.sSymbolType <> '' THEN
	sPayloadRcv := '';
		Lynus_Standards.GVL_Communicator.arrInterfaceInfoValueWriteTo[fbJsonRead.stInfoFromReceivedMessage.byReadWriteArrayNumber].bWriteNewValue := TRUE;
			Lynus_Standards.GVL_Communicator.arrInterfaceInfoValueWriteTo[fbJsonRead.stInfoFromReceivedMessage.byReadWriteArrayNumber].sFullSymbolName := fbJsonRead.stInfoFromReceivedMessage.sFullSymbolName;
				Lynus_Standards.GVL_Communicator.arrInterfaceInfoValueWriteTo[fbJsonRead.stInfoFromReceivedMessage.byReadWriteArrayNumber].sSymbolType := fbJsonRead.stInfoFromReceivedMessage.sSymbolType;
					Lynus_Standards.GVL_Communicator.arrInterfaceInfoValueWriteTo[fbJsonRead.stInfoFromReceivedMessage.byReadWriteArrayNumber].arrValue := fbJsonRead.stInfoFromReceivedMessage.arrValue;	
						Lynus_Standards.GVL_Communicator.arrInterfaceInfoValueWriteTo[fbJsonRead.stInfoFromReceivedMessage.byReadWriteArrayNumber].uiSizeArray := fbJsonRead.stInfoFromReceivedMessage.uiSizeArray;
END_IF
	IF fbJsonRead.bError THEN sPayloadRcv := ''; END_IF
	
//Data to ADS Write
IF Lynus_Standards.GVL_Communicator.byNumberOfReadWriteFunction >= 1 AND Lynus_Standards.GVL_Communicator.byNumberOfReadWriteFunction <= 10 THEN
	FOR byLPWriteInterface := 1 TO Lynus_Standards.GVL_Communicator.byNumberOfReadWriteFunction BY 1 DO 
		Lynus_Standards.GVL_Communicator.arrInterfaceInfoValueWriteTo[byLPWriteInterface].udiCountBuffer := fbMessageQueue.nQueuedMessages; 
	END_FOR
ELSE
	FOR byLPWriteInterface := 1 TO 10 BY 1 DO 
		Lynus_Standards.GVL_Communicator.arrInterfaceInfoValueWriteTo[byLPWriteInterface].udiCountBuffer := 0; 
	END_FOR
END_IF

//Outputs
bConnected := fbMqttClient.bConnected;
	hrErrorCode := fbMqttClient.hrErrorCode;
		eConnectionState := fbMqttClient.eConnectionState;

//Data to send the connected Flag to the GVL to enable all other Lynus Devices on PLC
Lynus_Standards.GVL_Communicator.bStateConnectionToEnableFunctions := bConnected;	

IF Lynus_Standards.GVL_Communicator.byNumberOfReadWriteFunction >= 1 AND Lynus_Standards.GVL_Communicator.byNumberOfReadWriteFunction <= 10 THEN
	FOR byLPWriteInterface := 1 TO Lynus_Standards.GVL_Communicator.byNumberOfReadWriteFunction BY 1 DO 
		Lynus_Standards.GVL_Communicator.arrInterfaceInfoValueWriteTo[byLPWriteInterface].bSendFunctionOK := bConnected; 
	END_FOR
ELSE
	FOR byLPWriteInterface := 1 TO 10 BY 1 DO 
		Lynus_Standards.GVL_Communicator.arrInterfaceInfoValueWriteTo[byLPWriteInterface].bSendFunctionOK := FALSE;
	END_FOR
END_IF		
		
IF fbMqttClient.bError OR fbJsonRead.bError OR fbGetTime.ERR THEN bError := TRUE; ELSE bError := FALSE; END_IF	

IF fbJsonRead.bError THEN eErrorMessage_Out := fbJsonRead.eErrorMessage_Out; END_IF
IF fbJsonWrite.bError THEN eErrorMessage_Out := fbJsonWrite.eErrorMessage_Out; END_IF

IF NOT fbJsonRead.bError AND NOT fbJsonWrite.bError THEN eErrorMessage_Out := eErrorMessage.eNoError; END_IF  

//Clear receive buffer, if the json string has the error too long
timError(IN:= fbJsonRead.bError AND NOT timError.Q, PT:= T#30S, Q=> , ET=> );
	
IF timError.Q THEN 
	sPayloadRcv := '';
		bReadOut := FALSE;
			fbMessageQueue.ResetQueue();
END_IF

END_FUNCTION_BLOCK

// ---- FBs/FB_Shelly_Pro1PM_Helper.TcPOU
FUNCTION_BLOCK FB_Shelly_Pro1PM_Helper
VAR_INPUT
	bSend			: BOOL;
	bSetOnP1		: BOOL;
	bSetOffP1		: BOOL;
END_VAR

VAR_IN_OUT
	fbClient		: FB_IotHttpClient;
END_VAR

VAR_OUTPUT
	bBusy			: BOOL;
	bError			: BOOL;
	bStateP1		: BOOL;
	lrapowerP1		: LREAL;
	lrvoltageP1		: LREAL;
	lraenergyP1		: LREAL;
	lrTemperatureP1	: LREAL;
END_VAR

VAR
	fbRequestSwitch0	: FB_IotHttpRequest;
	fbRequestSwitch1	: FB_IotHttpRequest;
	RisingEdge			: R_TRIG;
	RisingEdgeSetOnP1	: R_TRIG;
	RisingEdgeSetOffP1	: R_TRIG;
	fbJson				: FB_JsonDomParser;
	nState				: UDINT;
	timTimeout			: TON;
	tTimeOut			: TIME := T#2S;
	timTimeoutSwitch	: TON;
	tTimeOutSwitch		: TIME := T#5S;
	bGetContentResult	: BOOL;
	sContentS0			: STRING(511);
	
	bGetJsonResult		: BOOL;
	jsonDoc				: SJsonValue;
	jsonVal				: SJsonValue;
	
	nReqCount			: UDINT;	
	nResCount			: UDINT;
	nValidResCount		: UDINT;
	nErrCount			: UDINT;
	
	fbRequest2         : FB_IotHttpRequest;
	fbRequest3         : FB_IotHttpRequest;
	fbHeader            : FB_IotHttpHeaderFieldMap;
	fbHeader2            : FB_IotHttpHeaderFieldMap;
	
	sRealm	:	STRING(511);
	sPassword :	STRING(511) := ':sh3lly4ankerio2$$';
	snonce	:	STRING(511);
	scnonce	:	STRING(511);
	shash	: STRING(511);
	bhash	: BOOL;
	
	aData	: STRING(511);
	a_ha1	: ARRAY[0..31] OF BYTE;
	str_ha1 : STRING(511);
	str_Toha1   : STRING(511);
	udint_length_string : UDINT;
	
	a_ha2	: ARRAY[0..31] OF BYTE;
	str_ha2 : STRING(511);
	str_Toha2   : STRING(511);
	
	a_response	: ARRAY[0..31] OF BYTE;
	str_response : STRING(511);
	str_Toresponse   : STRING(511);

	str_authorization	: STRING(2048);
	
	sfincontent	: STRING(511);
	int_CountOffWrite: INT;
	int_CountOnWrite: INT;
	str_URI : STRING(50);
	int_Mode: INT;
	ton_Timeout: Ton;
	b_Done: BOOL;
	nState_Old: UDINT;
	int_ErrorCount: INT;
END_VAR

//Timer for Timeout
timTimeout(IN:= (nState = 1 AND bBusy) OR (nState = nState_Old AND bBusy), PT:= tTimeOut, Q=> , ET=> );
	IF timTimeout.Q THEN 
		nState := 0;
		bBusy := FALSE;
		bStateP1 := FALSE;
		lrapowerP1 := 0;
		lrvoltageP1 := 0;
		lraenergyP1 := 0;
		lrTemperatureP1 := 0;		
	END_IF
IF nState<> nState_old THEN
	nState_old := nState;
END_IF	
(*timTimeoutSwitch(IN:= bSetOnP1 OR bSetOffP1, PT:= tTimeOut, Q=> , ET=> );
	IF timTimeoutSwitch.Q THEN 
		bSetOnP1 := FALSE;
		bSetOffP1 := FALSE;
	END_IF
*)
IF bError THEN
	int_ErrorCount := int_ErrorCount+1;
	bError := FALSE;
END_IF

RisingEdge(CLK:= bSend );
RisingEdgeSetOnP1(CLK:= bSetOnP1 );
RisingEdgeSetOffP1(CLK:= bSetOffP1 );

CASE nState OF
	1:
		IF
			fbRequestSwitch0.SendRequest(sUri:=str_URI, fbClient:=fbClient, eRequestType:=ETcIotHttpRequestType.HTTP_Get, 0, 0, 0) THEN
			nState:= 2;
			nReqCount:= nReqCount+1;
		END_IF
	
	2:
		IF NOT fbRequestSwitch0.bBusy THEN
			bError:= TRUE;
			IF NOT fbRequestSwitch0.bError THEN
				bGetContentResult:= fbRequestSwitch0.GetHeaderField(pValue:= ADR(sContentS0), 
														 nValueSize:= SIZEOF(sContentS0), sField := 'WWW-Authenticate');
				IF fbRequestSwitch0.nStatusCode = 401 THEN
					bGetJsonResult:= FALSE;
						sRealm := sContentS0;
						sRealm := DELETE(sRealm, FIND(sRealm, 'realm') + 7, 0);
						sRealm := DELETE(sRealm, LEN(sRealm), FIND(sRealm, '"'));
						
						snonce := sContentS0;
						snonce := DELETE(snonce, FIND(snonce, 'nonce') + 7, 0);
						snonce := DELETE(snonce, LEN(snonce), FIND(snonce, '"'));
						
						scnonce := 'YmawvYzT';
					
						aData := sRealm;
						
						str_Toha1:=concat('admin:', sRealm);
						str_Toha1:=concat(str_Toha1, sPassword);
		 
						udint_length_string:= len2(ADR(str_Toha1));
						F_GenerateHashValue(E_HashMode.HASH_SHA256,ADR(str_Toha1),udint_length_string,ADR(a_ha1),32);
						
							str_ha1:=concat(byte_to_hexstr(a_ha1[0],2,TRUE),byte_to_hexstr(a_ha1[1],2,TRUE));
							str_ha1:=concat(str_ha1,byte_to_hexstr(a_ha1[2],2,TRUE));
							str_ha1:=concat(str_ha1,byte_to_hexstr(a_ha1[3],2,TRUE));
							str_ha1:=concat(str_ha1,byte_to_hexstr(a_ha1[4],2,TRUE));
							str_ha1:=concat(str_ha1,byte_to_hexstr(a_ha1[5],2,TRUE));
							str_ha1:=concat(str_ha1,byte_to_hexstr(a_ha1[6],2,TRUE));
							str_ha1:=concat(str_ha1,byte_to_hexstr(a_ha1[7],2,TRUE));
							str_ha1:=concat(str_ha1,byte_to_hexstr(a_ha1[8],2,TRUE));
							str_ha1:=concat(str_ha1,byte_to_hexstr(a_ha1[9],2,TRUE));
							str_ha1:=concat(str_ha1,byte_to_hexstr(a_ha1[10],2,TRUE));
							str_ha1:=concat(str_ha1,byte_to_hexstr(a_ha1[11],2,TRUE));
							str_ha1:=concat(str_ha1,byte_to_hexstr(a_ha1[12],2,TRUE));
							str_ha1:=concat(str_ha1,byte_to_hexstr(a_ha1[13],2,TRUE));
							str_ha1:=concat(str_ha1,byte_to_hexstr(a_ha1[14],2,TRUE));
							str_ha1:=concat(str_ha1,byte_to_hexstr(a_ha1[15],2,TRUE));
							str_ha1:=concat(str_ha1,byte_to_hexstr(a_ha1[16],2,TRUE));
							str_ha1:=concat(str_ha1,byte_to_hexstr(a_ha1[17],2,TRUE));
							str_ha1:=concat(str_ha1,byte_to_hexstr(a_ha1[18],2,TRUE));
							str_ha1:=concat(str_ha1,byte_to_hexstr(a_ha1[19],2,TRUE));
							str_ha1:=concat(str_ha1,byte_to_hexstr(a_ha1[20],2,TRUE));
							str_ha1:=concat(str_ha1,byte_to_hexstr(a_ha1[21],2,TRUE));
							str_ha1:=concat(str_ha1,byte_to_hexstr(a_ha1[22],2,TRUE));
							str_ha1:=concat(str_ha1,byte_to_hexstr(a_ha1[23],2,TRUE));
							str_ha1:=concat(str_ha1,byte_to_hexstr(a_ha1[24],2,TRUE));
							str_ha1:=concat(str_ha1,byte_to_hexstr(a_ha1[25],2,TRUE));
							str_ha1:=concat(str_ha1,byte_to_hexstr(a_ha1[26],2,TRUE));
							str_ha1:=concat(str_ha1,byte_to_hexstr(a_ha1[27],2,TRUE));
							str_ha1:=concat(str_ha1,byte_to_hexstr(a_ha1[28],2,TRUE));
							str_ha1:=concat(str_ha1,byte_to_hexstr(a_ha1[29],2,TRUE));
							str_ha1:=concat(str_ha1,byte_to_hexstr(a_ha1[30],2,TRUE));
							str_ha1:=concat(str_ha1,byte_to_hexstr(a_ha1[31],2,TRUE));
						
						str_Toha2:= concat('GET:',str_URI);
				 
						udint_length_string:= len2(ADR(str_Toha2));
						F_GenerateHashValue(E_HashMode.HASH_SHA256,ADR(str_Toha2),udint_length_string,ADR(a_ha2),32);
						
							str_ha2:=concat(byte_to_hexstr(a_ha2[0],2,TRUE),byte_to_hexstr(a_ha2[1],2,TRUE));
							str_ha2:=concat(str_ha2,byte_to_hexstr(a_ha2[2],2,TRUE));
							str_ha2:=concat(str_ha2,byte_to_hexstr(a_ha2[3],2,TRUE));
							str_ha2:=concat(str_ha2,byte_to_hexstr(a_ha2[4],2,TRUE));
							str_ha2:=concat(str_ha2,byte_to_hexstr(a_ha2[5],2,TRUE));
							str_ha2:=concat(str_ha2,byte_to_hexstr(a_ha2[6],2,TRUE));
							str_ha2:=concat(str_ha2,byte_to_hexstr(a_ha2[7],2,TRUE));
							str_ha2:=concat(str_ha2,byte_to_hexstr(a_ha2[8],2,TRUE));
							str_ha2:=concat(str_ha2,byte_to_hexstr(a_ha2[9],2,TRUE));
							str_ha2:=concat(str_ha2,byte_to_hexstr(a_ha2[10],2,TRUE));
							str_ha2:=concat(str_ha2,byte_to_hexstr(a_ha2[11],2,TRUE));
							str_ha2:=concat(str_ha2,byte_to_hexstr(a_ha2[12],2,TRUE));
							str_ha2:=concat(str_ha2,byte_to_hexstr(a_ha2[13],2,TRUE));
							str_ha2:=concat(str_ha2,byte_to_hexstr(a_ha2[14],2,TRUE));
							str_ha2:=concat(str_ha2,byte_to_hexstr(a_ha2[15],2,TRUE));
							str_ha2:=concat(str_ha2,byte_to_hexstr(a_ha2[16],2,TRUE));
							str_ha2:=concat(str_ha2,byte_to_hexstr(a_ha2[17],2,TRUE));
							str_ha2:=concat(str_ha2,byte_to_hexstr(a_ha2[18],2,TRUE));
							str_ha2:=concat(str_ha2,byte_to_hexstr(a_ha2[19],2,TRUE));
							str_ha2:=concat(str_ha2,byte_to_hexstr(a_ha2[20],2,TRUE));
							str_ha2:=concat(str_ha2,byte_to_hexstr(a_ha2[21],2,TRUE));
							str_ha2:=concat(str_ha2,byte_to_hexstr(a_ha2[22],2,TRUE));
							str_ha2:=concat(str_ha2,byte_to_hexstr(a_ha2[23],2,TRUE));
							str_ha2:=concat(str_ha2,byte_to_hexstr(a_ha2[24],2,TRUE));
							str_ha2:=concat(str_ha2,byte_to_hexstr(a_ha2[25],2,TRUE));
							str_ha2:=concat(str_ha2,byte_to_hexstr(a_ha2[26],2,TRUE));
							str_ha2:=concat(str_ha2,byte_to_hexstr(a_ha2[27],2,TRUE));
							str_ha2:=concat(str_ha2,byte_to_hexstr(a_ha2[28],2,TRUE));
							str_ha2:=concat(str_ha2,byte_to_hexstr(a_ha2[29],2,TRUE));
							str_ha2:=concat(str_ha2,byte_to_hexstr(a_ha2[30],2,TRUE));
							str_ha2:=concat(str_ha2,byte_to_hexstr(a_ha2[31],2,TRUE));
							
						// <ha1> + ":" + <nonce> + ":" + <nc> + ":" + <cnonce> + ":" + "auth" + ":" + <ha2>
						
						str_Toresponse:=concat(str_ha1,':');
						str_Toresponse:=concat(str_Toresponse,snonce);
						str_Toresponse:=concat(str_Toresponse,':00000001:');
						str_Toresponse:=concat(str_Toresponse,scnonce);
						str_Toresponse:=concat(str_Toresponse,':');
						str_Toresponse:=concat(str_Toresponse,'auth:');
						str_Toresponse:=concat(str_Toresponse,str_ha2);
						
						udint_length_string:= len2(ADR(str_Toresponse));
						F_GenerateHashValue(E_HashMode.HASH_SHA256,ADR(str_Toresponse),udint_length_string,ADR(a_response),32);
						
							str_response:=concat(byte_to_hexstr(a_response[0],2,TRUE),byte_to_hexstr(a_response[1],2,TRUE));
							str_response:=concat(str_response,byte_to_hexstr(a_response[2],2,TRUE));
							str_response:=concat(str_response,byte_to_hexstr(a_response[3],2,TRUE));
							str_response:=concat(str_response,byte_to_hexstr(a_response[4],2,TRUE));
							str_response:=concat(str_response,byte_to_hexstr(a_response[5],2,TRUE));
							str_response:=concat(str_response,byte_to_hexstr(a_response[6],2,TRUE));
							str_response:=concat(str_response,byte_to_hexstr(a_response[7],2,TRUE));
							str_response:=concat(str_response,byte_to_hexstr(a_response[8],2,TRUE));
							str_response:=concat(str_response,byte_to_hexstr(a_response[9],2,TRUE));
							str_response:=concat(str_response,byte_to_hexstr(a_response[10],2,TRUE));
							str_response:=concat(str_response,byte_to_hexstr(a_response[11],2,TRUE));
							str_response:=concat(str_response,byte_to_hexstr(a_response[12],2,TRUE));
							str_response:=concat(str_response,byte_to_hexstr(a_response[13],2,TRUE));
							str_response:=concat(str_response,byte_to_hexstr(a_response[14],2,TRUE));
							str_response:=concat(str_response,byte_to_hexstr(a_response[15],2,TRUE));
							str_response:=concat(str_response,byte_to_hexstr(a_response[16],2,TRUE));
							str_response:=concat(str_response,byte_to_hexstr(a_response[17],2,TRUE));
							str_response:=concat(str_response,byte_to_hexstr(a_response[18],2,TRUE));
							str_response:=concat(str_response,byte_to_hexstr(a_response[19],2,TRUE));
							str_response:=concat(str_response,byte_to_hexstr(a_response[20],2,TRUE));
							str_response:=concat(str_response,byte_to_hexstr(a_response[21],2,TRUE));
							str_response:=concat(str_response,byte_to_hexstr(a_response[22],2,TRUE));
							str_response:=concat(str_response,byte_to_hexstr(a_response[23],2,TRUE));
							str_response:=concat(str_response,byte_to_hexstr(a_response[24],2,TRUE));
							str_response:=concat(str_response,byte_to_hexstr(a_response[25],2,TRUE));
							str_response:=concat(str_response,byte_to_hexstr(a_response[26],2,TRUE));
							str_response:=concat(str_response,byte_to_hexstr(a_response[27],2,TRUE));
							str_response:=concat(str_response,byte_to_hexstr(a_response[28],2,TRUE));
							str_response:=concat(str_response,byte_to_hexstr(a_response[29],2,TRUE));
							str_response:=concat(str_response,byte_to_hexstr(a_response[30],2,TRUE));
							str_response:=concat(str_response,byte_to_hexstr(a_response[31],2,TRUE));
							
						// "Digest username=\"admin\", realm=\"shellypro3em-083af27cfbac\", nonce=\"63768368\", uri=\"/rpc/EM.GetStatus?id=0\", algorithm=\"SHA-256\", qop=auth, nc=00000001, cnonce=\"oKOklSrS\", response=\"d1d59d1e015dee0a3acfc97b20a0fa0ff851b03d79ca00df59ce018a63041468\""
						
						str_authorization:=concat('Digest username="admin", realm="',sRealm);
						str_authorization:=concat(str_authorization,'", nonce="');
						str_authorization:=concat(str_authorization,snonce);
						str_authorization:=concat(str_authorization,'", algorithm="SHA-256", uri="/rpc/EM.GetStatus?id=0\"');
						str_authorization:=concat(str_authorization,str_URI);
						str_authorization:=concat(str_authorization,'", qop=auth, nc=00000001, cnonce="');
						str_authorization:=concat(str_authorization,scnonce);
						str_authorization:=concat(str_authorization,'", response="');
						str_authorization:=concat(str_authorization,str_response);
						str_authorization:=concat(str_authorization,'"');
						
						fbHeader.AddField('Authorization', str_authorization, FALSE);
						IF fbRequest2.SendRequest(sUri:= str_URI, fbClient:= fbClient, eRequestType:= ETcIotHttpRequestType.HTTP_Get, 0, 0, fbHeader) THEN
							nState:= 3;
							bBusy:= TRUE;
							bError:= FALSE;
						END_IF
				END_IF
			END_IF
		END_IF
	
	3:
		IF NOT fbRequest2.bBusy THEN
			bError:= TRUE;
			IF int_Mode<>0 THEN
				bError:= FALSE;
			END_IF
			IF NOT fbRequest2.bError THEN		//AND int_Mode=0 				 
				bGetContentResult:= fbRequest2.GetContent(pContent:= ADR(sfincontent), nContentSize:= SIZEOF(sfincontent), bSetNullTermination:= TRUE);
	
				IF fbRequest2.nStatusCode >= 200 AND fbRequest2.nStatusCode < 300 THEN
					bGetJsonResult:= FALSE;
					jsonDoc:= fbRequest2.GetJsonDomContent(fbJson);
					IF jsonDoc <> 0 THEN
						bGetJsonResult:= TRUE;
						IF fbJson.HasMember(jsonDoc, 'output')  THEN
							jsonVal:= fbJson.FindMember(jsonDoc, 'output');
							nValidResCount:= nValidResCount+1;					
							IF fbJson.IsBool(jsonVal) AND (fbJson.GetBool(jsonVal)=TRUE OR fbJson.GetBool(jsonVal)=FALSE) THEN							
								bStateP1:= fbJson.GetBool(jsonVal);									
							END_IF
						END_IF
						IF fbJson.HasMember(jsonDoc, 'apower')  THEN
							jsonVal:= fbJson.FindMember(jsonDoc, 'apower');
							nValidResCount:= nValidResCount+1;
							IF fbJson.IsDouble(jsonVal) AND fbJson.GetDouble(jsonVal)> -3.402823E+38 AND fbJson.GetDouble(jsonVal)< 3.402823E+38 THEN							
								lrapowerP1:= fbJson.GetDouble(jsonVal);									
							END_IF
						END_IF
						IF fbJson.HasMember(jsonDoc, 'voltage')  THEN
							jsonVal:= fbJson.FindMember(jsonDoc, 'voltage');
							nValidResCount:= nValidResCount+1;					
							IF fbJson.IsDouble(jsonVal) AND fbJson.GetDouble(jsonVal)> -3.402823E+38 AND fbJson.GetDouble(jsonVal)< 3.402823E+38 THEN
								lrvoltageP1:= fbJson.GetDouble(jsonVal);									
							END_IF
						END_IF
						IF fbJson.HasMember(jsonDoc, 'temperature')  THEN
							jsonVal:= fbJson.FindMember(jsonDoc, 'temperature');
							 IF fbJson.HasMember(jsonVal, 'tC') AND fbJson.GetDouble(jsonVal)> -3.402823E+38 AND fbJson.GetDouble(jsonVal)< 3.402823E+38 THEN							
								jsonVal:= fbJson.FindMember(jsonVal, 'tC');
								nValidResCount:= nValidResCount+1;					
								IF fbJson.IsDouble(jsonVal) AND fbJson.GetDouble(jsonVal)> -3.402823E+38 AND fbJson.GetDouble(jsonVal)< 3.402823E+38 THEN
									lrTemperatureP1:= fbJson.GetDouble(jsonVal);									
								END_IF
							END_IF
						END_IF
						IF fbJson.HasMember(jsonDoc, 'aenergy')  THEN
							jsonVal:= fbJson.FindMember(jsonDoc, 'aenergy');
							IF fbJson.HasMember(jsonVal, 'total') AND fbJson.GetDouble(jsonVal)> -3.402823E+38 AND fbJson.GetDouble(jsonVal)< 3.402823E+38 THEN							
								jsonVal:= fbJson.FindMember(jsonVal, 'total');
								nValidResCount:= nValidResCount+1;
								IF fbJson.IsDouble(jsonVal) AND fbJson.GetDouble(jsonVal)> -3.402823E+38 AND fbJson.GetDouble(jsonVal)< 3.402823E+38 THEN
									lraenergyP1:= fbJson.GetDouble(jsonVal);
								END_IF
							bError:= FALSE;
							END_IF
						END_IF	
					nResCount:= nResCount+1;			
					END_IF
				END_IF
			END_IF
		nState:= 4;
//		bBusy:= FALSE;
			IF bError THEN
				nErrCount:= nErrCount+1;
			END_IF
		ELSE
			ton_Timeout.IN := TRUE;
			IF ton_Timeout.Q THEN
				nState:= 3;	
				ton_Timeout.IN := FALSE;
			END_IF
		END_IF
	
	
	4:
		ton_Timeout.IN := FALSE;
		nState:= 6;
		
	6:
		bBusy:= FALSE;
		nState:= 0;

	
END_CASE

ton_Timeout(PT := T#5S);

END_FUNCTION_BLOCK
